LIN {X 0,Y 297.256,Z 379.745,A -85,B 0,C 180,E1 -16418.721,E2 -16418.721} C_VEL
LIN {X 0,Y 296.722,Z 381.976,A -85,B 0,C 180,E1 -16420.719,E2 -16420.719} C_VEL
LIN {X 0,Y 296.34,Z 383.559,A -85,B 0,C 180,E1 -16423.451,E2 -16423.451} C_VEL
LIN {X 0,Y 296.213,Z 383.714,A -85,B 0,C 180,E1 -16425.377,E2 -16425.377} C_VEL
LIN {X 0,Y 296.21,Z 383.053,A -85,B 0,C 180,E1 -16427.348,E2 -16427.348} C_VEL
LIN {X 0,Y 296.316,Z 381.493,A -85,B 0,C 180,E1 -16429.371,E2 -16429.371} C_VEL
LIN {X 0,Y 296.789,Z 378.032,A -85,B 0,C 180,E1 -16432,E2 -16432} C_VEL
LIN {X 0,Y 297.171,Z 374.788,A -85,B 0,C 180,E1 -16433.756,E2 -16433.756} C_VEL
LIN {X 0,Y 297.824,Z 369.2,A -85,B 0,C 180,E1 -16436.076,E2 -16436.076} C_VEL
LIN {X 0,Y 298.573,Z 363.535,A -85,B 0,C 180,E1 -16437.925,E2 -16437.925} C_VEL
LIN {X 0,Y 299.623,Z 356.033,A -85,B 0,C 180,E1 -16439.912,E2 -16439.912} C_VEL
LIN {X 0,Y 300.83,Z 347.311,A -85,B 0,C 180,E1 -16441.766,E2 -16441.766} C_VEL
LIN {X 0,Y 302.031,Z 337.923,A -85,B 0,C 180,E1 -16443.39,E2 -16443.39} C_VEL
LIN {X 0,Y 303.358,Z 327.596,A -85,B 0,C 180,E1 -16444.836,E2 -16444.836} C_VEL
LIN {X 0,Y 304.461,Z 317.398,A -85,B 0,C 180,E1 -16445.994,E2 -16445.994} C_VEL
LIN {X 0,Y 304.418,Z 313.925,A -85,B 0,C 180,E1 -16446.352,E2 -16446.352} C_VEL
LIN {X 0,Y 302.572,Z 302.571,A -85,B 0,C 180,E1 -16447.465,E2 -16447.465} C_VEL
LIN {X 0,Y 299.904,Z 289.87,A -85,B 0,C 180,E1 -16448.477,E2 -16448.477} C_VEL
LIN {X 0,Y 297.33,Z 278.987,A -85,B 0,C 180,E1 -16449.189,E2 -16449.189} C_VEL
LIN {X 0,Y 297.572,Z 275.868,A -85,B 0,C 180,E1 -16452.12,E2 -16452.12} C_VEL
LIN {X 0,Y 297.966,Z 271.492,A -85,B 0,C 180,E1 -16456.358,E2 -16456.358} C_VEL
LIN {X 0,Y 298.352,Z 267.326,A -85,B 0,C 180,E1 -16460.509,E2 -16460.509} C_VEL
LIN {X 0,Y 298.55,Z 266.296,A -85,B 0,C 180,E1 -16461.619,E2 -16461.619} C_VEL
LIN {X 0,Y 298.625,Z 266.288,A -85,B 0,C 180,E1 -16464.599,E2 -16464.599} C_VEL
LIN {X 0,Y 298.915,Z 266.253,A -85,B 0,C 180,E1 -16468.653,E2 -16468.653} C_VEL
LIN {X 0,Y 298.918,Z 266.248,A -85,B 0,C 180,E1 -16471.347,E2 -16471.347} C_VEL
LIN {X 0,Y 298.651,Z 266.281,A -85,B 0,C 180,E1 -16475.401,E2 -16475.401} C_VEL
LIN {X 0,Y 298.749,Z 266.273,A -85,B 0,C 180,E1 -16478.114,E2 -16478.114} C_VEL
LIN {X 0,Y 298.546,Z 266.299,A -85,B 0,C 180,E1 -16482.232,E2 -16482.232} C_VEL
LIN {X 0,Y 298.596,Z 266.288,A -85,B 0,C 180,E1 -16485.209,E2 -16485.209} C_VEL
LIN {X 0,Y 298.533,Z 266.295,A -85,B 0,C 180,E1 -16489.243,E2 -16489.243} C_VEL
LIN {X 0,Y 298.455,Z 266.308,A -85,B 0,C 180,E1 -16493.598,E2 -16493.598} C_VEL
LIN {X 0,Y 298.48,Z 266.301,A -85,B 0,C 180,E1 -16496.575,E2 -16496.575} C_VEL
LIN {X 0,Y 298.412,Z 266.312,A -85,B 0,C 180,E1 -16499.642,E2 -16499.642} C_VEL
LIN {X 0,Y 298.388,Z 266.314,A -85,B 0,C 180,E1 -16502.801,E2 -16502.801} C_VEL
LIN {X 0,Y 298.461,Z 266.305,A -85,B 0,C 180,E1 -16506.815,E2 -16506.815} C_VEL
LIN {X 0,Y 298.447,Z 266.307,A -85,B 0,C 180,E1 -16511.25,E2 -16511.25} C_VEL
LIN {X 0,Y 298.48,Z 266.303,A -85,B 0,C 180,E1 -16515.062,E2 -16515.062} C_VEL
LIN {X 0,Y 298.444,Z 266.309,A -85,B 0,C 180,E1 -16518.899,E2 -16518.899} C_VEL
LIN {X 0,Y 298.457,Z 266.309,A -85,B 0,C 180,E1 -16523.189,E2 -16523.189} C_VEL
LIN {X 0,Y 298.387,Z 266.314,A -85,B 0,C 180,E1 -16527.201,E2 -16527.201} C_VEL
LIN {X 0,Y 298.424,Z 266.307,A -85,B 0,C 180,E1 -16530.616,E2 -16530.616} C_VEL
LIN {X 0,Y 298.476,Z 266.302,A -85,B 0,C 180,E1 -16533.476,E2 -16533.476} C_VEL
LIN {X 0,Y 298.428,Z 266.312,A -85,B 0,C 180,E1 -16536.699,E2 -16536.699} C_VEL
LIN {X 0,Y 298.532,Z 266.3,A -85,B 0,C 180,E1 -16540.758,E2 -16540.758} C_VEL
LIN {X 0,Y 298.587,Z 266.288,A -85,B 0,C 180,E1 -16544.996,E2 -16544.996} C_VEL
LIN {X 0,Y 298.585,Z 266.286,A -85,B 0,C 180,E1 -16549.148,E2 -16549.148} C_VEL
LIN {X 0,Y 298.735,Z 266.27,A -85,B 0,C 180,E1 -16551.887,E2 -16551.887} C_VEL
LIN {X 0,Y 298.752,Z 266.266,A -85,B 0,C 180,E1 -16552.865,E2 -16552.865} C_VEL
LIN {X 0,Y 298.15,Z 266.346,A -85,B 0,C 180,E1 -16553.989,E2 -16553.989} C_VEL
LIN {X 0,Y 295.364,Z 266.697,A -85,B 0,C 180,E1 -16555.82,E2 -16555.82} C_VEL
LIN {X 0,Y 292.977,Z 266.993,A -85,B 0,C 180,E1 -16557.306,E2 -16557.306} C_VEL
LIN {X 0,Y 291.962,Z 267.117,A -85,B 0,C 180,E1 -16558.456,E2 -16558.456} C_VEL
LIN {X 0,Y 291.886,Z 267.124,A -85,B 0,C 180,E1 -16558.845,E2 -16558.845} C_VEL
LIN {X 0,Y 291.886,Z 267.122,A -85,B 0,C 180,E1 -16561.381,E2 -16561.381} C_VEL
LIN {X 0,Y 291.743,Z 267.139,A -85,B 0,C 180,E1 -16566.92,E2 -16566.92} C_VEL
LIN {X 0,Y 291.627,Z 267.158,A -85,B 0,C 180,E1 -16569.714,E2 -16569.714} C_VEL
LIN {X 0,Y 291.52,Z 267.173,A -85,B 0,C 180,E1 -16573.952,E2 -16573.952} C_VEL
LIN {X 0,Y 291.485,Z 267.172,A -85,B 0,C 180,E1 -16576.82,E2 -16576.82} C_VEL
LIN {X 0,Y 291.45,Z 267.181,A -85,B 0,C 180,E1 -16579.876,E2 -16579.876} C_VEL
LIN {X 0,Y 291.398,Z 267.185,A -85,B 0,C 180,E1 -16584.207,E2 -16584.207} C_VEL
LIN {X 0,Y 291.418,Z 267.184,A -85,B 0,C 180,E1 -16587.273,E2 -16587.273} C_VEL
LIN {X 0,Y 291.334,Z 267.193,A -85,B 0,C 180,E1 -16590.439,E2 -16590.439} C_VEL
LIN {X 0,Y 291.345,Z 267.194,A -85,B 0,C 180,E1 -16593.7,E2 -16593.7} C_VEL
LIN {X 0,Y 291.378,Z 267.192,A -85,B 0,C 180,E1 -16597.256,E2 -16597.256} C_VEL
LIN {X 0,Y 291.335,Z 267.194,A -85,B 0,C 180,E1 -16600.644,E2 -16600.644} C_VEL
LIN {X 0,Y 291.292,Z 267.199,A -85,B 0,C 180,E1 -16604.403,E2 -16604.403} C_VEL
LIN {X 0,Y 291.364,Z 267.287,A -85,B 0,C 180,E1 -16605.706,E2 -16605.706} C_VEL
LIN {X 0,Y 292.179,Z 271.679,A -85,B 0,C 180,E1 -16609.5,E2 -16609.5} C_VEL
LIN {X 0,Y 292.693,Z 275.227,A -85,B 0,C 180,E1 -16612.41,E2 -16612.41} C_VEL
LIN {X 0,Y 292.739,Z 278.292,A -85,B 0,C 180,E1 -16614.818,E2 -16614.818} C_VEL
LIN {X 0,Y 292.076,Z 282.608,A -85,B 0,C 180,E1 -16618.038,E2 -16618.038} C_VEL
LIN {X 0,Y 291.167,Z 289.009,A -85,B 0,C 180,E1 -16622.703,E2 -16622.703} C_VEL
LIN {X 0,Y 290.666,Z 294.198,A -85,B 0,C 180,E1 -16626.394,E2 -16626.394} C_VEL
LIN {X 0,Y 293.234,Z 308.199,A -85,B 0,C 180,E1 -16627.253,E2 -16627.253} C_VEL
LIN {X 0,Y 295.062,Z 320.852,A -85,B 0,C 180,E1 -16628.271,E2 -16628.271} C_VEL
LIN {X 0,Y 296.269,Z 331.555,A -85,B 0,C 180,E1 -16629.338,E2 -16629.338} C_VEL
LIN {X 0,Y 296.691,Z 338.172,A -85,B 0,C 180,E1 -16630.092,E2 -16630.092} C_VEL
LIN {X 0,Y 295.207,Z 348.791,A -85,B 0,C 180,E1 -16631.433,E2 -16631.433} C_VEL
LIN {X 0,Y 293.834,Z 359.224,A -85,B 0,C 180,E1 -16633.087,E2 -16633.087} C_VEL
LIN {X 0,Y 292.498,Z 369.063,A -85,B 0,C 180,E1 -16635.031,E2 -16635.031} C_VEL
LIN {X 0,Y 291.312,Z 377.393,A -85,B 0,C 180,E1 -16637.105,E2 -16637.105} C_VEL
LIN {X 0,Y 290.47,Z 384.109,A -85,B 0,C 180,E1 -16639.192,E2 -16639.192} C_VEL
LIN {X 0,Y 289.851,Z 390.238,A -85,B 0,C 180,E1 -16641.635,E2 -16641.635} C_VEL
LIN {X 0,Y 289.559,Z 394.197,A -85,B 0,C 180,E1 -16643.729,E2 -16643.729} C_VEL
LIN {X 0,Y 289.435,Z 397.097,A -85,B 0,C 180,E1 -16645.822,E2 -16645.822} C_VEL
LIN {X 0,Y 289.463,Z 398.458,A -85,B 0,C 180,E1 -16647.217,E2 -16647.217} C_VEL
LIN {X 0,Y 289.419,Z 399.41,A -85,B 0,C 180,E1 -16648.608,E2 -16648.608} C_VEL
LIN {X 0,Y 289.438,Z 399.968,A -85,B 0,C 180,E1 -16650,E2 -16650} C_VEL
LIN {X 0,Y 289.409,Z 400.104,A -85,B 0,C 180,E1 -16651.391,E2 -16651.391} C_VEL
LIN {X 0,Y 289.432,Z 399.814,A -85,B 0,C 180,E1 -16652.783,E2 -16652.783} C_VEL
LIN {X 0,Y 289.481,Z 398.063,A -85,B 0,C 180,E1 -16655.573,E2 -16655.573} C_VEL
LIN {X 0,Y 289.638,Z 396.572,A -85,B 0,C 180,E1 -16656.968,E2 -16656.968} C_VEL
LIN {X 0,Y 290.082,Z 393.523,A -85,B 0,C 180,E1 -16659.06,E2 -16659.06} C_VEL
LIN {X 0,Y 290.789,Z 389.449,A -85,B 0,C 180,E1 -16661.148,E2 -16661.148} C_VEL
LIN {X 0,Y 292.006,Z 383.239,A -85,B 0,C 180,E1 -16663.571,E2 -16663.571} C_VEL
LIN {X 0,Y 293.614,Z 376.515,A -85,B 0,C 180,E1 -16665.621,E2 -16665.621} C_VEL
LIN {X 0,Y 295.014,Z 369.133,A -85,B 0,C 180,E1 -16667.467,E2 -16667.467} C_VEL
LIN {X 0,Y 296.963,Z 359.815,A -85,B 0,C 180,E1 -16669.349,E2 -16669.349} C_VEL
LIN {X 0,Y 299.12,Z 349.497,A -85,B 0,C 180,E1 -16670.996,E2 -16670.996} C_VEL
LIN {X 0,Y 300.497,Z 342.181,A -85,B 0,C 180,E1 -16671.975,E2 -16671.975} C_VEL
LIN {X 0,Y 300.225,Z 332.312,A -85,B 0,C 180,E1 -16673.273,E2 -16673.273} C_VEL
LIN {X 0,Y 299.063,Z 321.612,A -85,B 0,C 180,E1 -16674.529,E2 -16674.529} C_VEL
LIN {X 0,Y 297.128,Z 311.576,A -85,B 0,C 180,E1 -16675.605,E2 -16675.605} C_VEL
LIN {X 0,Y 293.476,Z 298.869,A -85,B 0,C 180,E1 -16676.88,E2 -16676.88} C_VEL
LIN {X 0,Y 291.642,Z 293.187,A -85,B 0,C 180,E1 -16677.401,E2 -16677.401} C_VEL
LIN {X 0,Y 291.589,Z 292.614,A -85,B 0,C 180,E1 -16677.494,E2 -16677.494} C_VEL
LIN {X 0,Y 292.14,Z 288.963,A -85,B 0,C 180,E1 -16680.343,E2 -16680.343} C_VEL
LIN {X 0,Y 292.807,Z 285.096,A -85,B 0,C 180,E1 -16683.507,E2 -16683.507} C_VEL
LIN {X 0,Y 293.161,Z 282.887,A -85,B 0,C 180,E1 -16685.402,E2 -16685.402} C_VEL
LIN {X 0,Y 293.236,Z 279.487,A -85,B 0,C 180,E1 -16688.545,E2 -16688.545} C_VEL
LIN {X 0,Y 292.811,Z 275.93,A -85,B 0,C 180,E1 -16692.224,E2 -16692.224} C_VEL
LIN {X 0,Y 292.299,Z 272.574,A -85,B 0,C 180,E1 -16696.162,E2 -16696.162} C_VEL
LIN {X 0,Y 291.787,Z 269.447,A -85,B 0,C 180,E1 -16700.42,E2 -16700.42} C_VEL
LIN {X 0,Y 291.524,Z 267.869,A -85,B 0,C 180,E1 -16702.935,E2 -16702.935} C_VEL
LIN {X 0,Y 291.389,Z 267.189,A -85,B 0,C 180,E1 -16705.087,E2 -16705.087} C_VEL
LIN {X 0,Y 291.371,Z 267.192,A -85,B 0,C 180,E1 -16707.949,E2 -16707.949} C_VEL
LIN {X 0,Y 291.38,Z 267.189,A -85,B 0,C 180,E1 -16711.157,E2 -16711.157} C_VEL
LIN {X 0,Y 291.415,Z 267.187,A -85,B 0,C 180,E1 -16714.27,E2 -16714.27} C_VEL
LIN {X 0,Y 291.378,Z 267.19,A -85,B 0,C 180,E1 -16717.298,E2 -16717.298} C_VEL
LIN {X 0,Y 291.455,Z 267.181,A -85,B 0,C 180,E1 -16720.268,E2 -16720.268} C_VEL
LIN {X 0,Y 291.537,Z 267.172,A -85,B 0,C 180,E1 -16724.633,E2 -16724.633} C_VEL
LIN {X 0,Y 291.532,Z 267.171,A -85,B 0,C 180,E1 -16728.879,E2 -16728.879} C_VEL
LIN {X 0,Y 291.704,Z 267.151,A -85,B 0,C 180,E1 -16731.687,E2 -16731.687} C_VEL
LIN {X 0,Y 291.625,Z 267.158,A -85,B 0,C 180,E1 -16734.467,E2 -16734.467} C_VEL
LIN {X 0,Y 291.884,Z 267.126,A -85,B 0,C 180,E1 -16738.619,E2 -16738.619} C_VEL
LIN {X 0,Y 292.013,Z 267.48,A -85,B 0,C 180,E1 -16739.998,E2 -16739.998} C_VEL
LIN {X 0,Y 292.074,Z 269.02,A -85,B 0,C 180,E1 -16742.757,E2 -16742.757} C_VEL
LIN {X 0,Y 292.277,Z 271.603,A -85,B 0,C 180,E1 -16746.904,E2 -16746.904} C_VEL
LIN {X 0,Y 292.339,Z 273.56,A -85,B 0,C 180,E1 -16749.722,E2 -16749.722} C_VEL
LIN {X 0,Y 291.837,Z 276.856,A -85,B 0,C 180,E1 -16753.933,E2 -16753.933} C_VEL
LIN {X 0,Y 291.452,Z 279.266,A -85,B 0,C 180,E1 -16756.818,E2 -16756.818} C_VEL
LIN {X 0,Y 291.228,Z 280.798,A -85,B 0,C 180,E1 -16758.6,E2 -16758.6} C_VEL
LIN {X 0,Y 292.241,Z 283.889,A -85,B 0,C 180,E1 -16758.897,E2 -16758.897} C_VEL
LIN {X 0,Y 296.303,Z 294.553,A -85,B 0,C 180,E1 -16760.086,E2 -16760.086} C_VEL
LIN {X 0,Y 299.322,Z 304.767,A -85,B 0,C 180,E1 -16761.272,E2 -16761.272} C_VEL
LIN {X 0,Y 301.593,Z 316.345,A -85,B 0,C 180,E1 -16762.716,E2 -16762.716} C_VEL
LIN {X 0,Y 302.352,Z 322.44,A -85,B 0,C 180,E1 -16763.539,E2 -16763.539} C_VEL
LIN {X 0,Y 300.502,Z 333.167,A -85,B 0,C 180,E1 -16764.894,E2 -16764.894} C_VEL
LIN {X 0,Y 298.4,Z 343.82,A -85,B 0,C 180,E1 -16766.581,E2 -16766.581} C_VEL
LIN {X 0,Y 296.514,Z 352.555,A -85,B 0,C 180,E1 -16768.295,E2 -16768.295} C_VEL
LIN {X 0,Y 294.957,Z 359.715,A -85,B 0,C 180,E1 -16770.022,E2 -16770.022} C_VEL
LIN {X 0,Y 293.128,Z 367.333,A -85,B 0,C 180,E1 -16772.313,E2 -16772.313} C_VEL
LIN {X 0,Y 291.934,Z 372.454,A -85,B 0,C 180,E1 -16774.268,E2 -16774.268} C_VEL
LIN {X 0,Y 291.015,Z 376.512,A -85,B 0,C 180,E1 -16776.223,E2 -16776.223} C_VEL
LIN {X 0,Y 290.349,Z 379.544,A -85,B 0,C 180,E1 -16778.112,E2 -16778.112} C_VEL
LIN {X 0,Y 290.043,Z 380.865,A -85,B 0,C 180,E1 -16779.161,E2 -16779.161} C_VEL
LIN {X 0,Y 289.559,Z 382.745,A -85,B 0,C 180,E1 -16781.202,E2 -16781.202} C_VEL
LIN {X 0,Y 289.272,Z 383.745,A -85,B 0,C 180,E1 -16783.21,E2 -16783.21} C_VEL
LIN {X 0,Y 289.136,Z 383.93,A -85,B 0,C 180,E1 -16785.18,E2 -16785.18} C_VEL
LIN {X 0,Y 289.1,Z 383.357,A -85,B 0,C 180,E1 -16787.105,E2 -16787.105} C_VEL
LIN {X 0,Y 289.291,Z 381.069,A -85,B 0,C 180,E1 -16789.926,E2 -16789.926} C_VEL
LIN {X 0,Y 289.666,Z 378.543,A -85,B 0,C 180,E1 -16791.836,E2 -16791.836} C_VEL
LIN {X 0,Y 290.236,Z 373.662,A -85,B 0,C 180,E1 -16794.469,E2 -16794.469} C_VEL
LIN {X 0,Y 290.917,Z 368.352,A -85,B 0,C 180,E1 -16796.596,E2 -16796.596} C_VEL
LIN {X 0,Y 291.897,Z 361.234,A -85,B 0,C 180,E1 -16798.826,E2 -16798.826} C_VEL
LIN {X 0,Y 293.127,Z 352.689,A -85,B 0,C 180,E1 -16800.955,E2 -16800.955} C_VEL
LIN {X 0,Y 294.342,Z 343.846,A -85,B 0,C 180,E1 -16802.724,E2 -16802.724} C_VEL
LIN {X 0,Y 295.724,Z 333.278,A -85,B 0,C 180,E1 -16804.427,E2 -16804.427} C_VEL
LIN {X 0,Y 297.002,Z 323.285,A -85,B 0,C 180,E1 -16805.724,E2 -16805.724} C_VEL
LIN {X 0,Y 297.663,Z 316.026,A -85,B 0,C 180,E1 -16806.521,E2 -16806.521} C_VEL
LIN {X 0,Y 295.95,Z 304.983,A -85,B 0,C 180,E1 -16807.67,E2 -16807.67} C_VEL
LIN {X 0,Y 293.272,Z 291.758,A -85,B 0,C 180,E1 -16808.796,E2 -16808.796} C_VEL
LIN {X 0,Y 290.272,Z 279.187,A -85,B 0,C 180,E1 -16809.633,E2 -16809.633} C_VEL
LIN {X 0,Y 290.557,Z 275.578,A -85,B 0,C 180,E1 -16813.127,E2 -16813.127} C_VEL
LIN {X 0,Y 290.879,Z 272.648,A -85,B 0,C 180,E1 -16816.019,E2 -16816.019} C_VEL
LIN {X 0,Y 291.278,Z 268.444,A -85,B 0,C 180,E1 -16820.277,E2 -16820.277} C_VEL
LIN {X 0,Y 291.504,Z 267.174,A -85,B 0,C 180,E1 -16821.683,E2 -16821.683} C_VEL
LIN {X 0,Y 291.59,Z 267.163,A -85,B 0,C 180,E1 -16824.468,E2 -16824.468} C_VEL
LIN {X 0,Y 291.881,Z 267.129,A -85,B 0,C 180,E1 -16828.621,E2 -16828.621} C_VEL
LIN {X 0,Y 291.884,Z 267.124,A -85,B 0,C 180,E1 -16831.38,E2 -16831.38} C_VEL
LIN {X 0,Y 291.736,Z 267.144,A -85,B 0,C 180,E1 -16836.918,E2 -16836.918} C_VEL
LIN {X 0,Y 291.62,Z 267.158,A -85,B 0,C 180,E1 -16839.712,E2 -16839.712} C_VEL
LIN {X 0,Y 291.513,Z 267.173,A -85,B 0,C 180,E1 -16843.951,E2 -16843.951} C_VEL
LIN {X 0,Y 291.477,Z 267.174,A -85,B 0,C 180,E1 -16846.818,E2 -16846.818} C_VEL
LIN {X 0,Y 291.442,Z 267.182,A -85,B 0,C 180,E1 -16849.876,E2 -16849.876} C_VEL
LIN {X 0,Y 291.413,Z 267.185,A -85,B 0,C 180,E1 -16854.204,E2 -16854.204} C_VEL
LIN {X 0,Y 291.413,Z 267.181,A -85,B 0,C 180,E1 -16857.272,E2 -16857.272} C_VEL
LIN {X 0,Y 291.329,Z 267.193,A -85,B 0,C 180,E1 -16860.437,E2 -16860.437} C_VEL
LIN {X 0,Y 291.336,Z 267.197,A -85,B 0,C 180,E1 -16863.699,E2 -16863.699} C_VEL
LIN {X 0,Y 291.396,Z 267.187,A -85,B 0,C 180,E1 -16867.262,E2 -16867.262} C_VEL
LIN {X 0,Y 291.397,Z 267.181,A -85,B 0,C 180,E1 -16870.631,E2 -16870.631} C_VEL
LIN {X 0,Y 291.397,Z 267.182,A -85,B 0,C 180,E1 -16874.38,E2 -16874.38} C_VEL
LIN {X 0,Y 291.38,Z 267.187,A -85,B 0,C 180,E1 -16878.392,E2 -16878.392} C_VEL
LIN {X 0,Y 291.371,Z 267.192,A -85,B 0,C 180,E1 -16881.164,E2 -16881.164} C_VEL
LIN {X 0,Y 291.377,Z 267.187,A -85,B 0,C 180,E1 -16884.631,E2 -16884.631} C_VEL
LIN {X 0,Y 291.363,Z 267.184,A -85,B 0,C 180,E1 -16887.952,E2 -16887.952} C_VEL
LIN {X 0,Y 291.375,Z 267.188,A -85,B 0,C 180,E1 -16891.16,E2 -16891.16} C_VEL
LIN {X 0,Y 291.409,Z 267.182,A -85,B 0,C 180,E1 -16894.273,E2 -16894.273} C_VEL
LIN {X 0,Y 291.374,Z 267.189,A -85,B 0,C 180,E1 -16897.301,E2 -16897.301} C_VEL
LIN {X 0,Y 291.451,Z 267.179,A -85,B 0,C 180,E1 -16900.272,E2 -16900.272} C_VEL
LIN {X 0,Y 291.534,Z 267.169,A -85,B 0,C 180,E1 -16904.636,E2 -16904.636} C_VEL
LIN {X 0,Y 291.529,Z 267.166,A -85,B 0,C 180,E1 -16908.882,E2 -16908.882} C_VEL
LIN {X 0,Y 291.682,Z 267.147,A -85,B 0,C 180,E1 -16911.689,E2 -16911.689} C_VEL
LIN {X 0,Y 291.622,Z 267.161,A -85,B 0,C 180,E1 -16914.47,E2 -16914.47} C_VEL
LIN {X 0,Y 291.886,Z 267.124,A -85,B 0,C 180,E1 -16918.845,E2 -16918.845} C_VEL
LIN {X 0,Y 291.563,Z 267.164,A -85,B 0,C 180,E1 -16919.616,E2 -16919.616} C_VEL
LIN {X 0,Y 289.526,Z 267.419,A -85,B 0,C 180,E1 -16921.126,E2 -16921.126} C_VEL
LIN {X 0,Y 285.64,Z 267.9,A -85,B 0,C 180,E1 -16923.39,E2 -16923.39} C_VEL
LIN {X 0,Y 284.593,Z 268.028,A -85,B 0,C 180,E1 -16924.573,E2 -16924.573} C_VEL
LIN {X 0,Y 284.53,Z 268.034,A -85,B 0,C 180,E1 -16924.973,E2 -16924.973} C_VEL
LIN {X 0,Y 284.695,Z 268.016,A -85,B 0,C 180,E1 -16927.092,E2 -16927.092} C_VEL
LIN {X 0,Y 284.565,Z 268.039,A -85,B 0,C 180,E1 -16929.957,E2 -16929.957} C_VEL
LIN {X 0,Y 284.477,Z 268.048,A -85,B 0,C 180,E1 -16934.305,E2 -16934.305} C_VEL
LIN {X 0,Y 284.423,Z 268.052,A -85,B 0,C 180,E1 -16937.25,E2 -16937.25} C_VEL
LIN {X 0,Y 284.378,Z 268.059,A -85,B 0,C 180,E1 -16940.244,E2 -16940.244} C_VEL
LIN {X 0,Y 284.368,Z 268.063,A -85,B 0,C 180,E1 -16943.876,E2 -16943.876} C_VEL
LIN {X 0,Y 284.394,Z 268.058,A -85,B 0,C 180,E1 -16947.174,E2 -16947.174} C_VEL
LIN {X 0,Y 284.294,Z 268.073,A -85,B 0,C 180,E1 -16951.276,E2 -16951.276} C_VEL
LIN {X 0,Y 284.342,Z 268.067,A -85,B 0,C 180,E1 -16955.349,E2 -16955.349} C_VEL
LIN {X 0,Y 284.314,Z 268.068,A -85,B 0,C 180,E1 -16958.17,E2 -16958.17} C_VEL
LIN {X 0,Y 284.271,Z 268.073,A -85,B 0,C 180,E1 -16962.126,E2 -16962.126} C_VEL
LIN {X 0,Y 284.318,Z 268.271,A -85,B 0,C 180,E1 -16965.577,E2 -16965.577} C_VEL
LIN {X 0,Y 284.93,Z 271.255,A -85,B 0,C 180,E1 -16968.244,E2 -16968.244} C_VEL
LIN {X 0,Y 285.603,Z 275.711,A -85,B 0,C 180,E1 -16972.035,E2 -16972.035} C_VEL
LIN {X 0,Y 285.72,Z 278.465,A -85,B 0,C 180,E1 -16974.266,E2 -16974.266} C_VEL
LIN {X 0,Y 285.222,Z 282.234,A -85,B 0,C 180,E1 -16977.174,E2 -16977.174} C_VEL
LIN {X 0,Y 284.22,Z 288.642,A -85,B 0,C 180,E1 -16981.978,E2 -16981.978} C_VEL
LIN {X 0,Y 283.649,Z 294.031,A -85,B 0,C 180,E1 -16985.918,E2 -16985.918} C_VEL
LIN {X 0,Y 286.123,Z 307.348,A -85,B 0,C 180,E1 -16986.745,E2 -16986.745} C_VEL
LIN {X 0,Y 288.089,Z 320.565,A -85,B 0,C 180,E1 -16987.838,E2 -16987.838} C_VEL
LIN {X 0,Y 289.345,Z 331.936,A -85,B 0,C 180,E1 -16989.006,E2 -16989.006} C_VEL
LIN {X 0,Y 289.749,Z 338.469,A -85,B 0,C 180,E1 -16989.779,E2 -16989.779} C_VEL
LIN {X 0,Y 288.104,Z 350.156,A -85,B 0,C 180,E1 -16991.327,E2 -16991.327} C_VEL
LIN {X 0,Y 286.817,Z 359.652,A -85,B 0,C 180,E1 -16992.9,E2 -16992.9} C_VEL
LIN {X 0,Y 285.606,Z 368.348,A -85,B 0,C 180,E1 -16994.661,E2 -16994.661} C_VEL
LIN {X 0,Y 284.371,Z 376.786,A -85,B 0,C 180,E1 -16996.785,E2 -16996.785} C_VEL
LIN {X 0,Y 283.462,Z 383.575,A -85,B 0,C 180,E1 -16998.922,E2 -16998.922} C_VEL
LIN {X 0,Y 282.799,Z 389.798,A -85,B 0,C 180,E1 -17001.425,E2 -17001.425} C_VEL
LIN {X 0,Y 282.492,Z 393.817,A -85,B 0,C 180,E1 -17003.572,E2 -17003.572} C_VEL
LIN {X 0,Y 282.342,Z 396.767,A -85,B 0,C 180,E1 -17005.717,E2 -17005.717} C_VEL
LIN {X 0,Y 282.369,Z 398.165,A -85,B 0,C 180,E1 -17007.147,E2 -17007.147} C_VEL
LIN {X 0,Y 282.342,Z 399.144,A -85,B 0,C 180,E1 -17008.573,E2 -17008.573} C_VEL
LIN {X 0,Y 282.358,Z 399.727,A -85,B 0,C 180,E1 -17010,E2 -17010} C_VEL
LIN {X 0,Y 282.333,Z 399.908,A -85,B 0,C 180,E1 -17011.426,E2 -17011.426} C_VEL
LIN {X 0,Y 282.338,Z 399.648,A -85,B 0,C 180,E1 -17012.853,E2 -17012.853} C_VEL
LIN {X 0,Y 282.391,Z 397.95,A -85,B 0,C 180,E1 -17015.713,E2 -17015.713} C_VEL
LIN {X 0,Y 282.579,Z 396.51,A -85,B 0,C 180,E1 -17017.143,E2 -17017.143} C_VEL
LIN {X 0,Y 283.057,Z 393.517,A -85,B 0,C 180,E1 -17019.287,E2 -17019.287} C_VEL
LIN {X 0,Y 283.816,Z 389.503,A -85,B 0,C 180,E1 -17021.425,E2 -17021.425} C_VEL
LIN {X 0,Y 285.108,Z 383.389,A -85,B 0,C 180,E1 -17023.906,E2 -17023.906} C_VEL
LIN {X 0,Y 286.796,Z 376.739,A -85,B 0,C 180,E1 -17026.002,E2 -17026.002} C_VEL
LIN {X 0,Y 288.634,Z 367.851,A -85,B 0,C 180,E1 -17028.261,E2 -17028.261} C_VEL
LIN {X 0,Y 290.753,Z 358.408,A -85,B 0,C 180,E1 -17030.147,E2 -17030.147} C_VEL
LIN {X 0,Y 293.043,Z 347.904,A -85,B 0,C 180,E1 -17031.822,E2 -17031.822} C_VEL
LIN {X 0,Y 294.002,Z 341.921,A -85,B 0,C 180,E1 -17032.649,E2 -17032.649} C_VEL
LIN {X 0,Y 293.528,Z 330.262,A -85,B 0,C 180,E1 -17034.213,E2 -17034.213} C_VEL
LIN {X 0,Y 291.859,Z 317.94,A -85,B 0,C 180,E1 -17035.685,E2 -17035.685} C_VEL
LIN {X 0,Y 288.827,Z 305.475,A -85,B 0,C 180,E1 -17037.078,E2 -17037.078} C_VEL
LIN {X 0,Y 285.489,Z 295.291,A -85,B 0,C 180,E1 -17038.136,E2 -17038.136} C_VEL
LIN {X 0,Y 284.738,Z 292.405,A -85,B 0,C 180,E1 -17038.407,E2 -17038.407} C_VEL
LIN {X 0,Y 285.639,Z 287.112,A -85,B 0,C 180,E1 -17042.771,E2 -17042.771} C_VEL
LIN {X 0,Y 286.199,Z 283.326,A -85,B 0,C 180,E1 -17046.11,E2 -17046.11} C_VEL
LIN {X 0,Y 286.277,Z 281.113,A -85,B 0,C 180,E1 -17048.223,E2 -17048.223} C_VEL
LIN {X 0,Y 285.913,Z 277.91,A -85,B 0,C 180,E1 -17051.58,E2 -17051.58} C_VEL
LIN {X 0,Y 285.426,Z 274.532,A -85,B 0,C 180,E1 -17055.565,E2 -17055.565} C_VEL
LIN {X 0,Y 284.915,Z 271.383,A -85,B 0,C 180,E1 -17059.877,E2 -17059.877} C_VEL
LIN {X 0,Y 284.52,Z 269.091,A -85,B 0,C 180,E1 -17063.64,E2 -17063.64} C_VEL
LIN {X 0,Y 284.34,Z 268.198,A -85,B 0,C 180,E1 -17065.353,E2 -17065.353} C_VEL
LIN {X 0,Y 284.294,Z 268.072,A -85,B 0,C 180,E1 -17068.724,E2 -17068.724} C_VEL
LIN {X 0,Y 284.396,Z 268.06,A -85,B 0,C 180,E1 -17072.825,E2 -17072.825} C_VEL
LIN {X 0,Y 284.364,Z 268.065,A -85,B 0,C 180,E1 -17076.705,E2 -17076.705} C_VEL
LIN {X 0,Y 284.4,Z 268.059,A -85,B 0,C 180,E1 -17081.26,E2 -17081.26} C_VEL
LIN {X 0,Y 284.474,Z 268.052,A -85,B 0,C 180,E1 -17084.468,E2 -17084.468} C_VEL
LIN {X 0,Y 284.484,Z 268.05,A -85,B 0,C 180,E1 -17088.6,E2 -17088.6} C_VEL
LIN {X 0,Y 284.654,Z 268.029,A -85,B 0,C 180,E1 -17091.479,E2 -17091.479} C_VEL
LIN {X 0,Y 284.596,Z 268.034,A -85,B 0,C 180,E1 -17094.33,E2 -17094.33} C_VEL
LIN {X 0,Y 284.739,Z 268.017,A -85,B 0,C 180,E1 -17097.169,E2 -17097.169} C_VEL
LIN {X 0,Y 284.883,Z 268.286,A -85,B 0,C 180,E1 -17098.585,E2 -17098.585} C_VEL
LIN {X 0,Y 285.12,Z 269.678,A -85,B 0,C 180,E1 -17101.411,E2 -17101.411} C_VEL
LIN {X 0,Y 285.278,Z 272.935,A -85,B 0,C 180,E1 -17106.908,E2 -17106.908} C_VEL
LIN {X 0,Y 285.327,Z 274.985,A -85,B 0,C 180,E1 -17109.927,E2 -17109.927} C_VEL
LIN {X 0,Y 284.973,Z 277.165,A -85,B 0,C 180,E1 -17112.822,E2 -17112.822} C_VEL
LIN {X 0,Y 284.599,Z 279.509,A -85,B 0,C 180,E1 -17115.76,E2 -17115.76} C_VEL
LIN {X 0,Y 284.327,Z 281.063,A -85,B 0,C 180,E1 -17117.624,E2 -17117.624} C_VEL
LIN {X 0,Y 285.381,Z 284.267,A -85,B 0,C 180,E1 -17117.973,E2 -17117.973} C_VEL
LIN {X 0,Y 289.433,Z 294.425,A -85,B 0,C 180,E1 -17119.18,E2 -17119.18} C_VEL
LIN {X 0,Y 292.846,Z 305.93,A -85,B 0,C 180,E1 -17120.602,E2 -17120.602} C_VEL
LIN {X 0,Y 295.002,Z 316.877,A -85,B 0,C 180,E1 -17122.036,E2 -17122.036} C_VEL
LIN {X 0,Y 295.819,Z 324.286,A -85,B 0,C 180,E1 -17123.077,E2 -17123.077} C_VEL
LIN {X 0,Y 293.719,Z 335.646,A -85,B 0,C 180,E1 -17124.601,E2 -17124.601} C_VEL
LIN {X 0,Y 291.696,Z 345.269,A -85,B 0,C 180,E1 -17126.211,E2 -17126.211} C_VEL
LIN {X 0,Y 289.567,Z 354.379,A -85,B 0,C 180,E1 -17128.114,E2 -17128.114} C_VEL
LIN {X 0,Y 287.808,Z 361.793,A -85,B 0,C 180,E1 -17130.037,E2 -17130.037} C_VEL
LIN {X 0,Y 286.035,Z 368.807,A -85,B 0,C 180,E1 -17132.301,E2 -17132.301} C_VEL
LIN {X 0,Y 284.694,Z 374.307,A -85,B 0,C 180,E1 -17134.593,E2 -17134.593} C_VEL
LIN {X 0,Y 283.85,Z 377.755,A -85,B 0,C 180,E1 -17136.455,E2 -17136.455} C_VEL
LIN {X 0,Y 283.187,Z 380.448,A -85,B 0,C 180,E1 -17138.345,E2 -17138.345} C_VEL
LIN {X 0,Y 282.634,Z 382.441,A -85,B 0,C 180,E1 -17140.277,E2 -17140.277} C_VEL
LIN {X 0,Y 282.306,Z 383.686,A -85,B 0,C 180,E1 -17142.231,E2 -17142.231} C_VEL
LIN {X 0,Y 282.075,Z 384.16,A -85,B 0,C 180,E1 -17144.234,E2 -17144.234} C_VEL
LIN {X 0,Y 282.012,Z 383.853,A -85,B 0,C 180,E1 -17146.275,E2 -17146.275} C_VEL
LIN {X 0,Y 282.029,Z 382.69,A -85,B 0,C 180,E1 -17148.378,E2 -17148.378} C_VEL
LIN {X 0,Y 282.291,Z 380.595,A -85,B 0,C 180,E1 -17150.511,E2 -17150.511} C_VEL
LIN {X 0,Y 282.729,Z 377.437,A -85,B 0,C 180,E1 -17152.694,E2 -17152.694} C_VEL
LIN {X 0,Y 283.382,Z 372.369,A -85,B 0,C 180,E1 -17155.222,E2 -17155.222} C_VEL
LIN {X 0,Y 284.226,Z 365.982,A -85,B 0,C 180,E1 -17157.637,E2 -17157.637} C_VEL
LIN {X 0,Y 285.184,Z 359.408,A -85,B 0,C 180,E1 -17159.598,E2 -17159.598} C_VEL
LIN {X 0,Y 286.473,Z 350.732,A -85,B 0,C 180,E1 -17161.678,E2 -17161.678} C_VEL
LIN {X 0,Y 287.798,Z 341.157,A -85,B 0,C 180,E1 -17163.535,E2 -17163.535} C_VEL
LIN {X 0,Y 289.112,Z 331.728,A -85,B 0,C 180,E1 -17165.017,E2 -17165.017} C_VEL
LIN {X 0,Y 290.539,Z 320.094,A -85,B 0,C 180,E1 -17166.478,E2 -17166.478} C_VEL
LIN {X 0,Y 290.778,Z 316.872,A -85,B 0,C 180,E1 -17166.837,E2 -17166.837} C_VEL
LIN {X 0,Y 289.04,Z 305.673,A -85,B 0,C 180,E1 -17168.048,E2 -17168.048} C_VEL
LIN {X 0,Y 286.385,Z 292.575,A -85,B 0,C 180,E1 -17169.208,E2 -17169.208} C_VEL
LIN {X 0,Y 283.246,Z 279.387,A -85,B 0,C 180,E1 -17170.108,E2 -17170.108} C_VEL
LIN {X 0,Y 283.591,Z 275.274,A -85,B 0,C 180,E1 -17174.181,E2 -17174.181} C_VEL
LIN {X 0,Y 283.887,Z 272.39,A -85,B 0,C 180,E1 -17177.127,E2 -17177.127} C_VEL
LIN {X 0,Y 284.46,Z 268.052,A -85,B 0,C 180,E1 -17181.717,E2 -17181.717} C_VEL
LIN {X 0,Y 284.554,Z 268.038,A -85,B 0,C 180,E1 -17184.331,E2 -17184.331} C_VEL
LIN {X 0,Y 284.847,Z 268.006,A -85,B 0,C 180,E1 -17188.586,E2 -17188.586} C_VEL
LIN {X 0,Y 284.85,Z 268.001,A -85,B 0,C 180,E1 -17191.414,E2 -17191.414} C_VEL
LIN {X 0,Y 284.688,Z 268.022,A -85,B 0,C 180,E1 -17197.09,E2 -17197.09} C_VEL
LIN {X 0,Y 284.557,Z 268.039,A -85,B 0,C 180,E1 -17199.956,E2 -17199.956} C_VEL
LIN {X 0,Y 284.472,Z 268.051,A -85,B 0,C 180,E1 -17204.303,E2 -17204.303} C_VEL
LIN {X 0,Y 284.416,Z 268.053,A -85,B 0,C 180,E1 -17207.249,E2 -17207.249} C_VEL
LIN {X 0,Y 284.372,Z 268.063,A -85,B 0,C 180,E1 -17210.243,E2 -17210.243} C_VEL
LIN {X 0,Y 284.375,Z 268.064,A -85,B 0,C 180,E1 -17213.883,E2 -17213.883} C_VEL
LIN {X 0,Y 284.388,Z 268.056,A -85,B 0,C 180,E1 -17217.174,E2 -17217.174} C_VEL
LIN {X 0,Y 284.288,Z 268.07,A -85,B 0,C 180,E1 -17221.275,E2 -17221.275} C_VEL
LIN {X 0,Y 284.353,Z 268.065,A -85,B 0,C 180,E1 -17225.355,E2 -17225.355} C_VEL
LIN {X 0,Y 284.328,Z 268.064,A -85,B 0,C 180,E1 -17228.166,E2 -17228.166} C_VEL
LIN {X 0,Y 284.335,Z 268.059,A -85,B 0,C 180,E1 -17232.142,E2 -17232.142} C_VEL
LIN {X 0,Y 284.344,Z 268.062,A -85,B 0,C 180,E1 -17236.209,E2 -17236.209} C_VEL
LIN {X 0,Y 284.343,Z 268.064,A -85,B 0,C 180,E1 -17240.014,E2 -17240.014} C_VEL
LIN {X 0,Y 284.344,Z 268.063,A -85,B 0,C 180,E1 -17243.618,E2 -17243.618} C_VEL
LIN {X 0,Y 284.299,Z 268.067,A -85,B 0,C 180,E1 -17247.191,E2 -17247.191} C_VEL
LIN {X 0,Y 284.351,Z 268.056,A -85,B 0,C 180,E1 -17250.377,E2 -17250.377} C_VEL
LIN {X 0,Y 284.37,Z 268.059,A -85,B 0,C 180,E1 -17253.588,E2 -17253.588} C_VEL
LIN {X 0,Y 284.359,Z 268.065,A -85,B 0,C 180,E1 -17256.708,E2 -17256.708} C_VEL
LIN {X 0,Y 284.397,Z 268.057,A -85,B 0,C 180,E1 -17261.263,E2 -17261.263} C_VEL
LIN {X 0,Y 284.472,Z 268.048,A -85,B 0,C 180,E1 -17264.471,E2 -17264.471} C_VEL
LIN {X 0,Y 284.481,Z 268.044,A -85,B 0,C 180,E1 -17268.603,E2 -17268.603} C_VEL
LIN {X 0,Y 284.633,Z 268.024,A -85,B 0,C 180,E1 -17271.482,E2 -17271.482} C_VEL
LIN {X 0,Y 284.592,Z 268.036,A -85,B 0,C 180,E1 -17274.333,E2 -17274.333} C_VEL
LIN {X 0,Y 284.85,Z 268.001,A -85,B 0,C 180,E1 -17278.848,E2 -17278.848} C_VEL
LIN {X 0,Y 284.852,Z 267.998,A -85,B 0,C 180,E1 -17281.415,E2 -17281.415} C_VEL
LIN {X 0,Y 284.53,Z 268.034,A -85,B 0,C 180,E1 -17284.973,E2 -17284.973} C_VEL
LIN {X 0,Y 283.919,Z 268.116,A -85,B 0,C 180,E1 -17286.157,E2 -17286.157} C_VEL
LIN {X 0,Y 281.064,Z 268.474,A -85,B 0,C 180,E1 -17288.085,E2 -17288.085} C_VEL
LIN {X 0,Y 278.597,Z 268.78,A -85,B 0,C 180,E1 -17289.65,E2 -17289.65} C_VEL
LIN {X 0,Y 277.526,Z 268.913,A -85,B 0,C 180,E1 -17290.864,E2 -17290.864} C_VEL
LIN {X 0,Y 277.435,Z 268.924,A -85,B 0,C 180,E1 -17291.276,E2 -17291.276} C_VEL
LIN {X 0,Y 277.434,Z 268.927,A -85,B 0,C 180,E1 -17295.718,E2 -17295.718} C_VEL
LIN {X 0,Y 277.344,Z 268.934,A -85,B 0,C 180,E1 -17300.351,E2 -17300.351} C_VEL
LIN {X 0,Y 277.318,Z 268.94,A -85,B 0,C 180,E1 -17304.171,E2 -17304.171} C_VEL
LIN {X 0,Y 277.323,Z 268.94,A -85,B 0,C 180,E1 -17307.505,E2 -17307.505} C_VEL
LIN {X 0,Y 277.273,Z 268.945,A -85,B 0,C 180,E1 -17310.483,E2 -17310.483} C_VEL
LIN {X 0,Y 277.248,Z 268.948,A -85,B 0,C 180,E1 -17313.897,E2 -17313.897} C_VEL
LIN {X 0,Y 277.27,Z 268.949,A -85,B 0,C 180,E1 -17317.471,E2 -17317.471} C_VEL
LIN {X 0,Y 277.212,Z 268.956,A -85,B 0,C 180,E1 -17321.238,E2 -17321.238} C_VEL
LIN {X 0,Y 277.246,Z 269.006,A -85,B 0,C 180,E1 -17325.219,E2 -17325.219} C_VEL
LIN {X 0,Y 278.087,Z 273.505,A -85,B 0,C 180,E1 -17329.306,E2 -17329.306} C_VEL
LIN {X 0,Y 278.52,Z 275.988,A -85,B 0,C 180,E1 -17331.468,E2 -17331.468} C_VEL
LIN {X 0,Y 278.62,Z 279.688,A -85,B 0,C 180,E1 -17334.539,E2 -17334.539} C_VEL
LIN {X 0,Y 277.972,Z 284.005,A -85,B 0,C 180,E1 -17337.931,E2 -17337.931} C_VEL
LIN {X 0,Y 276.988,Z 290.395,A -85,B 0,C 180,E1 -17342.825,E2 -17342.825} C_VEL
LIN {X 0,Y 276.637,Z 293.857,A -85,B 0,C 180,E1 -17345.427,E2 -17345.427} C_VEL
LIN {X 0,Y 279.198,Z 307.438,A -85,B 0,C 180,E1 -17346.299,E2 -17346.299} C_VEL
LIN {X 0,Y 281.166,Z 320.847,A -85,B 0,C 180,E1 -17347.44,E2 -17347.44} C_VEL
LIN {X 0,Y 282.409,Z 332.312,A -85,B 0,C 180,E1 -17348.657,E2 -17348.657} C_VEL
LIN {X 0,Y 282.68,Z 340.162,A -85,B 0,C 180,E1 -17349.631,E2 -17349.631} C_VEL
LIN {X 0,Y 280.974,Z 351.515,A -85,B 0,C 180,E1 -17351.214,E2 -17351.214} C_VEL
LIN {X 0,Y 279.578,Z 361.385,A -85,B 0,C 180,E1 -17352.957,E2 -17352.957} C_VEL
LIN {X 0,Y 278.468,Z 369.171,A -85,B 0,C 180,E1 -17354.633,E2 -17354.633} C_VEL
LIN {X 0,Y 277.225,Z 377.418,A -85,B 0,C 180,E1 -17356.811,E2 -17356.811} C_VEL
LIN {X 0,Y 276.318,Z 384.058,A -85,B 0,C 180,E1 -17359.003,E2 -17359.003} C_VEL
LIN {X 0,Y 275.738,Z 389.339,A -85,B 0,C 180,E1 -17361.203,E2 -17361.203} C_VEL
LIN {X 0,Y 275.41,Z 393.421,A -85,B 0,C 180,E1 -17363.406,E2 -17363.406} C_VEL
LIN {X 0,Y 275.253,Z 396.419,A -85,B 0,C 180,E1 -17365.607,E2 -17365.607} C_VEL
LIN {X 0,Y 275.277,Z 397.868,A -85,B 0,C 180,E1 -17367.073,E2 -17367.073} C_VEL
LIN {X 0,Y 275.268,Z 398.874,A -85,B 0,C 180,E1 -17368.537,E2 -17368.537} C_VEL
LIN {X 0,Y 275.28,Z 399.483,A -85,B 0,C 180,E1 -17370,E2 -17370} C_VEL
LIN {X 0,Y 275.258,Z 399.697,A -85,B 0,C 180,E1 -17371.463,E2 -17371.463} C_VEL
LIN {X 0,Y 275.247,Z 399.487,A -85,B 0,C 180,E1 -17372.927,E2 -17372.927} C_VEL
LIN {X 0,Y 275.306,Z 397.848,A -85,B 0,C 180,E1 -17375.86,E2 -17375.86} C_VEL
LIN {X 0,Y 275.514,Z 396.441,A -85,B 0,C 180,E1 -17377.327,E2 -17377.327} C_VEL
LIN {X 0,Y 276.014,Z 393.503,A -85,B 0,C 180,E1 -17379.526,E2 -17379.526} C_VEL
LIN {X 0,Y 276.851,Z 389.552,A -85,B 0,C 180,E1 -17381.717,E2 -17381.717} C_VEL
LIN {X 0,Y 277.972,Z 384.498,A -85,B 0,C 180,E1 -17383.897,E2 -17383.897} C_VEL
LIN {X 0,Y 279.675,Z 378.212,A -85,B 0,C 180,E1 -17386.046,E2 -17386.046} C_VEL
LIN {X 0,Y 281.101,Z 371.971,A -85,B 0,C 180,E1 -17387.797,E2 -17387.797} C_VEL
LIN {X 0,Y 282.824,Z 364.258,A -85,B 0,C 180,E1 -17389.6,E2 -17389.6} C_VEL
LIN {X 0,Y 285.24,Z 354.08,A -85,B 0,C 180,E1 -17391.5,E2 -17391.5} C_VEL
LIN {X 0,Y 287.435,Z 343.836,A -85,B 0,C 180,E1 -17393.029,E2 -17393.029} C_VEL
LIN {X 0,Y 287.212,Z 333.033,A -85,B 0,C 180,E1 -17394.581,E2 -17394.581} C_VEL
LIN {X 0,Y 286.07,Z 322.519,A -85,B 0,C 180,E1 -17395.948,E2 -17395.948} C_VEL
LIN {X 0,Y 283.803,Z 311.278,A -85,B 0,C 180,E1 -17397.301,E2 -17397.301} C_VEL
LIN {X 0,Y 279.94,Z 298.502,A -85,B 0,C 180,E1 -17398.756,E2 -17398.756} C_VEL
LIN {X 0,Y 278.007,Z 292.928,A -85,B 0,C 180,E1 -17399.356,E2 -17399.356} C_VEL
LIN {X 0,Y 277.874,Z 292.176,A -85,B 0,C 180,E1 -17399.419,E2 -17399.419} C_VEL
LIN {X 0,Y 278.812,Z 287.188,A -85,B 0,C 180,E1 -17403.711,E2 -17403.711} C_VEL
LIN {X 0,Y 279.258,Z 283.485,A -85,B 0,C 180,E1 -17407.156,E2 -17407.156} C_VEL
LIN {X 0,Y 279.232,Z 281.664,A -85,B 0,C 180,E1 -17408.992,E2 -17408.992} C_VEL
LIN {X 0,Y 278.792,Z 278.169,A -85,B 0,C 180,E1 -17412.892,E2 -17412.892} C_VEL
LIN {X 0,Y 278.295,Z 274.922,A -85,B 0,C 180,E1 -17417.01,E2 -17417.01} C_VEL
LIN {X 0,Y 277.862,Z 272.383,A -85,B 0,C 180,E1 -17420.776,E2 -17420.776} C_VEL
LIN {X 0,Y 277.532,Z 270.334,A -85,B 0,C 180,E1 -17424.376,E2 -17424.376} C_VEL
LIN {X 0,Y 277.244,Z 268.951,A -85,B 0,C 180,E1 -17427.835,E2 -17427.835} C_VEL
LIN {X 0,Y 277.288,Z 268.944,A -85,B 0,C 180,E1 -17431.211,E2 -17431.211} C_VEL
LIN {X 0,Y 277.312,Z 268.943,A -85,B 0,C 180,E1 -17434.478,E2 -17434.478} C_VEL
LIN {X 0,Y 277.282,Z 268.946,A -85,B 0,C 180,E1 -17437.653,E2 -17437.653} C_VEL
LIN {X 0,Y 277.342,Z 268.94,A -85,B 0,C 180,E1 -17440.764,E2 -17440.764} C_VEL
LIN {X 0,Y 277.424,Z 268.928,A -85,B 0,C 180,E1 -17445.324,E2 -17445.324} C_VEL
LIN {X 0,Y 277.502,Z 268.919,A -85,B 0,C 180,E1 -17449.787,E2 -17449.787} C_VEL
LIN {X 0,Y 277.648,Z 268.902,A -85,B 0,C 180,E1 -17452.727,E2 -17452.727} C_VEL
LIN {X 0,Y 277.72,Z 269.177,A -85,B 0,C 180,E1 -17457.097,E2 -17457.097} C_VEL
LIN {X 0,Y 278.134,Z 270.421,A -85,B 0,C 180,E1 -17459.998,E2 -17459.998} C_VEL
LIN {X 0,Y 278.148,Z 271.93,A -85,B 0,C 180,E1 -17462.895,E2 -17462.895} C_VEL
LIN {X 0,Y 278.323,Z 274.495,A -85,B 0,C 180,E1 -17467.251,E2 -17467.251} C_VEL
LIN {X 0,Y 278.299,Z 276.44,A -85,B 0,C 180,E1 -17470.18,E2 -17470.18} C_VEL
LIN {X 0,Y 277.707,Z 279.796,A -85,B 0,C 180,E1 -17474.657,E2 -17474.657} C_VEL
LIN {X 0,Y 277.435,Z 281.337,A -85,B 0,C 180,E1 -17476.603,E2 -17476.603} C_VEL
LIN {X 0,Y 278.499,Z 284.479,A -85,B 0,C 180,E1 -17476.946,E2 -17476.946} C_VEL
LIN {X 0,Y 281.861,Z 292.418,A -85,B 0,C 180,E1 -17477.971,E2 -17477.971} C_VEL
LIN {X 0,Y 285.486,Z 303.581,A -85,B 0,C 180,E1 -17479.409,E2 -17479.409} C_VEL
LIN {X 0,Y 287.796,Z 313.338,A -85,B 0,C 180,E1 -17480.736,E2 -17480.736} C_VEL
LIN {X 0,Y 289.249,Z 323.378,A -85,B 0,C 180,E1 -17482.197,E2 -17482.197} C_VEL
LIN {X 0,Y 289.141,Z 326.916,A -85,B 0,C 180,E1 -17482.697,E2 -17482.697} C_VEL
LIN {X 0,Y 287.047,Z 337.544,A -85,B 0,C 180,E1 -17484.209,E2 -17484.209} C_VEL
LIN {X 0,Y 284.782,Z 347.446,A -85,B 0,C 180,E1 -17485.977,E2 -17485.977} C_VEL
LIN {X 0,Y 282.697,Z 355.948,A -85,B 0,C 180,E1 -17487.861,E2 -17487.861} C_VEL
LIN {X 0,Y 280.655,Z 363.881,A -85,B 0,C 180,E1 -17490.053,E2 -17490.053} C_VEL
LIN {X 0,Y 278.912,Z 370.292,A -85,B 0,C 180,E1 -17492.313,E2 -17492.313} C_VEL
LIN {X 0,Y 277.523,Z 375.599,A -85,B 0,C 180,E1 -17494.733,E2 -17494.733} C_VEL
LIN {X 0,Y 276.348,Z 380.178,A -85,B 0,C 180,E1 -17497.613,E2 -17497.613} C_VEL
LIN {X 0,Y 275.581,Z 382.719,A -85,B 0,C 180,E1 -17500.088,E2 -17500.088} C_VEL
LIN {X 0,Y 275.209,Z 383.985,A -85,B 0,C 180,E1 -17502.222,E2 -17502.222} C_VEL
LIN {X 0,Y 274.971,Z 384.388,A -85,B 0,C 180,E1 -17504.305,E2 -17504.305} C_VEL
LIN {X 0,Y 274.91,Z 383.987,A -85,B 0,C 180,E1 -17506.352,E2 -17506.352} C_VEL
LIN {X 0,Y 274.938,Z 382.86,A -85,B 0,C 180,E1 -17508.348,E2 -17508.348} C_VEL
LIN {X 0,Y 275.163,Z 381.015,A -85,B 0,C 180,E1 -17510.319,E2 -17510.319} C_VEL
LIN {X 0,Y 275.55,Z 378.398,A -85,B 0,C 180,E1 -17512.258,E2 -17512.258} C_VEL
LIN {X 0,Y 276.09,Z 374.292,A -85,B 0,C 180,E1 -17514.541,E2 -17514.541} C_VEL
LIN {X 0,Y 276.823,Z 368.717,A -85,B 0,C 180,E1 -17516.905,E2 -17516.905} C_VEL
LIN {X 0,Y 277.882,Z 361.403,A -85,B 0,C 180,E1 -17519.302,E2 -17519.302} C_VEL
LIN {X 0,Y 279.147,Z 353.277,A -85,B 0,C 180,E1 -17521.423,E2 -17521.423} C_VEL
LIN {X 0,Y 280.567,Z 343.586,A -85,B 0,C 180,E1 -17523.445,E2 -17523.445} C_VEL
LIN {X 0,Y 282.006,Z 333.509,A -85,B 0,C 180,E1 -17525.132,E2 -17525.132} C_VEL
LIN {X 0,Y 283.478,Z 322.361,A -85,B 0,C 180,E1 -17526.63,E2 -17526.63} C_VEL
LIN {X 0,Y 283.932,Z 318.606,A -85,B 0,C 180,E1 -17527.056,E2 -17527.056} C_VEL
LIN {X 0,Y 282.4,Z 307.938,A -85,B 0,C 180,E1 -17528.274,E2 -17528.274} C_VEL
LIN {X 0,Y 279.945,Z 295.282,A -85,B 0,C 180,E1 -17529.464,E2 -17529.464} C_VEL
LIN {X 0,Y 276.642,Z 281.552,A -85,B 0,C 180,E1 -17530.484,E2 -17530.484} C_VEL
LIN {X 0,Y 276.256,Z 279.563,A -85,B 0,C 180,E1 -17530.63,E2 -17530.63} C_VEL
LIN {X 0,Y 276.689,Z 274.973,A -85,B 0,C 180,E1 -17535.286,E2 -17535.286} C_VEL
LIN {X 0,Y 277.117,Z 270.701,A -85,B 0,C 180,E1 -17539.775,E2 -17539.775} C_VEL
LIN {X 0,Y 277.417,Z 268.929,A -85,B 0,C 180,E1 -17541.794,E2 -17541.794} C_VEL
LIN {X 0,Y 277.518,Z 268.914,A -85,B 0,C 180,E1 -17544.186,E2 -17544.186} C_VEL
LIN {X 0,Y 277.813,Z 268.881,A -85,B 0,C 180,E1 -17548.551,E2 -17548.551} C_VEL
LIN {X 0,Y 277.815,Z 268.877,A -85,B 0,C 180,E1 -17551.45,E2 -17551.45} C_VEL
LIN {X 0,Y 277.643,Z 268.899,A -85,B 0,C 180,E1 -17557.271,E2 -17557.271} C_VEL
LIN {X 0,Y 277.497,Z 268.92,A -85,B 0,C 180,E1 -17560.212,E2 -17560.212} C_VEL
LIN {X 0,Y 277.425,Z 268.927,A -85,B 0,C 180,E1 -17564.675,E2 -17564.675} C_VEL
LIN {X 0,Y 277.337,Z 268.935,A -85,B 0,C 180,E1 -17569.234,E2 -17569.234} C_VEL
LIN {X 0,Y 277.334,Z 268.941,A -85,B 0,C 180,E1 -17573.92,E2 -17573.92} C_VEL
LIN {X 0,Y 277.316,Z 268.938,A -85,B 0,C 180,E1 -17577.506,E2 -17577.506} C_VEL
LIN {X 0,Y 277.262,Z 268.944,A -85,B 0,C 180,E1 -17580.482,E2 -17580.482} C_VEL
LIN {X 0,Y 277.245,Z 268.951,A -85,B 0,C 180,E1 -17583.895,E2 -17583.895} C_VEL
LIN {X 0,Y 277.282,Z 268.946,A -85,B 0,C 180,E1 -17587.466,E2 -17587.466} C_VEL
LIN {X 0,Y 277.285,Z 268.94,A -85,B 0,C 180,E1 -17591.222,E2 -17591.222} C_VEL
LIN {X 0,Y 277.279,Z 268.943,A -85,B 0,C 180,E1 -17595.209,E2 -17595.209} C_VEL
LIN {X 0,Y 277.287,Z 268.946,A -85,B 0,C 180,E1 -17599.496,E2 -17599.496} C_VEL
LIN {X 0,Y 277.278,Z 268.944,A -85,B 0,C 180,E1 -17602.535,E2 -17602.535} C_VEL
LIN {X 0,Y 277.246,Z 268.943,A -85,B 0,C 180,E1 -17606.107,E2 -17606.107} C_VEL
LIN {X 0,Y 277.254,Z 268.94,A -85,B 0,C 180,E1 -17609.54,E2 -17609.54} C_VEL
LIN {X 0,Y 277.352,Z 268.934,A -85,B 0,C 180,E1 -17612.866,E2 -17612.866} C_VEL
LIN {X 0,Y 277.321,Z 268.938,A -85,B 0,C 180,E1 -17616.081,E2 -17616.081} C_VEL
LIN {X 0,Y 277.338,Z 268.94,A -85,B 0,C 180,E1 -17620.768,E2 -17620.768} C_VEL
LIN {X 0,Y 277.422,Z 268.92,A -85,B 0,C 180,E1 -17625.327,E2 -17625.327} C_VEL
LIN {X 0,Y 277.456,Z 268.915,A -85,B 0,C 180,E1 -17629.789,E2 -17629.789} C_VEL
LIN {X 0,Y 277.635,Z 268.9,A -85,B 0,C 180,E1 -17632.73,E2 -17632.73} C_VEL
LIN {X 0,Y 277.817,Z 268.878,A -85,B 0,C 180,E1 -17638.552,E2 -17638.552} C_VEL
LIN {X 0,Y 277.818,Z 268.874,A -85,B 0,C 180,E1 -17641.451,E2 -17641.451} C_VEL
LIN {X 0,Y 277.65,Z 268.894,A -85,B 0,C 180,E1 -17647.273,E2 -17647.273} C_VEL
LIN {X 0,Y 277.505,Z 268.918,A -85,B 0,C 180,E1 -17650.213,E2 -17650.213} C_VEL
LIN {X 0,Y 277.435,Z 268.924,A -85,B 0,C 180,E1 -17651.276,E2 -17651.276} C_VEL
LIN {X 0,Y 276.747,Z 269.013,A -85,B 0,C 180,E1 -17652.488,E2 -17652.488} C_VEL
LIN {X 0,Y 273.853,Z 269.37,A -85,B 0,C 180,E1 -17654.462,E2 -17654.462} C_VEL
LIN {X 0,Y 271.407,Z 269.675,A -85,B 0,C 180,E1 -17656.067,E2 -17656.067} C_VEL
LIN {X 0,Y 270.363,Z 269.803,A -85,B 0,C 180,E1 -17657.311,E2 -17657.311} C_VEL
LIN {X 0,Y 270.28,Z 269.81,A -85,B 0,C 180,E1 -17657.733,E2 -17657.733} C_VEL
LIN {X 0,Y 270.221,Z 269.823,A -85,B 0,C 180,E1 -17661.355,E2 -17661.355} C_VEL
LIN {X 0,Y 270.274,Z 269.816,A -85,B 0,C 180,E1 -17664.587,E2 -17664.587} C_VEL
LIN {X 0,Y 270.27,Z 269.816,A -85,B 0,C 180,E1 -17667.91,E2 -17667.91} C_VEL
LIN {X 0,Y 270.185,Z 269.832,A -85,B 0,C 180,E1 -17671.35,E2 -17671.35} C_VEL
LIN {X 0,Y 270.203,Z 269.827,A -85,B 0,C 180,E1 -17674.907,E2 -17674.907} C_VEL
LIN {X 0,Y 270.2,Z 269.827,A -85,B 0,C 180,E1 -17678.712,E2 -17678.712} C_VEL
LIN {X 0,Y 270.174,Z 269.83,A -85,B 0,C 180,E1 -17682.56,E2 -17682.56} C_VEL
LIN {X 0,Y 270.202,Z 269.907,A -85,B 0,C 180,E1 -17685.013,E2 -17685.013} C_VEL
LIN {X 0,Y 270.957,Z 273.942,A -85,B 0,C 180,E1 -17688.783,E2 -17688.783} C_VEL
LIN {X 0,Y 271.484,Z 277.074,A -85,B 0,C 180,E1 -17691.59,E2 -17691.59} C_VEL
LIN {X 0,Y 271.584,Z 280.369,A -85,B 0,C 180,E1 -17694.392,E2 -17694.392} C_VEL
LIN {X 0,Y 270.92,Z 284.68,A -85,B 0,C 180,E1 -17697.874,E2 -17697.874} C_VEL
LIN {X 0,Y 269.986,Z 290.261,A -85,B 0,C 180,E1 -17702.261,E2 -17702.261} C_VEL
LIN {X 0,Y 269.619,Z 293.681,A -85,B 0,C 180,E1 -17704.904,E2 -17704.904} C_VEL
LIN {X 0,Y 272.196,Z 307.18,A -85,B 0,C 180,E1 -17705.807,E2 -17705.807} C_VEL
LIN {X 0,Y 274.097,Z 320.505,A -85,B 0,C 180,E1 -17706.972,E2 -17706.972} C_VEL
LIN {X 0,Y 275.449,Z 332.578,A -85,B 0,C 180,E1 -17708.295,E2 -17708.295} C_VEL
LIN {X 0,Y 275.783,Z 340.327,A -85,B 0,C 180,E1 -17709.293,E2 -17709.293} C_VEL
LIN {X 0,Y 274.041,Z 351.608,A -85,B 0,C 180,E1 -17710.914,E2 -17710.914} C_VEL
LIN {X 0,Y 272.57,Z 361.52,A -85,B 0,C 180,E1 -17712.722,E2 -17712.722} C_VEL
LIN {X 0,Y 271.333,Z 369.905,A -85,B 0,C 180,E1 -17714.604,E2 -17714.604} C_VEL
LIN {X 0,Y 270.059,Z 377.988,A -85,B 0,C 180,E1 -17716.838,E2 -17716.838} C_VEL
LIN {X 0,Y 269.319,Z 383.474,A -85,B 0,C 180,E1 -17718.713,E2 -17718.713} C_VEL
LIN {X 0,Y 268.699,Z 388.83,A -85,B 0,C 180,E1 -17720.971,E2 -17720.971} C_VEL
LIN {X 0,Y 268.334,Z 392.982,A -85,B 0,C 180,E1 -17723.231,E2 -17723.231} C_VEL
LIN {X 0,Y 268.166,Z 396.048,A -85,B 0,C 180,E1 -17725.49,E2 -17725.49} C_VEL
LIN {X 0,Y 268.187,Z 397.556,A -85,B 0,C 180,E1 -17726.996,E2 -17726.996} C_VEL
LIN {X 0,Y 268.194,Z 398.597,A -85,B 0,C 180,E1 -17728.498,E2 -17728.498} C_VEL
LIN {X 0,Y 268.204,Z 399.236,A -85,B 0,C 180,E1 -17730,E2 -17730} C_VEL
LIN {X 0,Y 268.184,Z 399.479,A -85,B 0,C 180,E1 -17731.501,E2 -17731.501} C_VEL
LIN {X 0,Y 268.158,Z 399.322,A -85,B 0,C 180,E1 -17733.004,E2 -17733.004} C_VEL
LIN {X 0,Y 268.231,Z 397.745,A -85,B 0,C 180,E1 -17736.016,E2 -17736.016} C_VEL
LIN {X 0,Y 268.455,Z 396.368,A -85,B 0,C 180,E1 -17737.521,E2 -17737.521} C_VEL
LIN {X 0,Y 268.991,Z 393.496,A -85,B 0,C 180,E1 -17739.777,E2 -17739.777} C_VEL
LIN {X 0,Y 269.875,Z 389.627,A -85,B 0,C 180,E1 -17742.024,E2 -17742.024} C_VEL
LIN {X 0,Y 271.077,Z 384.665,A -85,B 0,C 180,E1 -17744.258,E2 -17744.258} C_VEL
LIN {X 0,Y 272.876,Z 378.463,A -85,B 0,C 180,E1 -17746.457,E2 -17746.457} C_VEL
LIN {X 0,Y 274.475,Z 371.501,A -85,B 0,C 180,E1 -17748.477,E2 -17748.477} C_VEL
LIN {X 0,Y 276.599,Z 363.067,A -85,B 0,C 180,E1 -17750.448,E2 -17750.448} C_VEL
LIN {X 0,Y 279.209,Z 352.652,A -85,B 0,C 180,E1 -17752.377,E2 -17752.377} C_VEL
LIN {X 0,Y 280.943,Z 344.729,A -85,B 0,C 180,E1 -17753.593,E2 -17753.593} C_VEL
LIN {X 0,Y 280.792,Z 334.266,A -85,B 0,C 180,E1 -17755.181,E2 -17755.181} C_VEL
LIN {X 0,Y 279.714,Z 323.575,A -85,B 0,C 180,E1 -17756.642,E2 -17756.642} C_VEL
LIN {X 0,Y 277.166,Z 311.267,A -85,B 0,C 180,E1 -17758.227,E2 -17758.227} C_VEL
LIN {X 0,Y 273.564,Z 299.235,A -85,B 0,C 180,E1 -17759.695,E2 -17759.695} C_VEL
LIN {X 0,Y 271.172,Z 292.555,A -85,B 0,C 180,E1 -17760.465,E2 -17760.465} C_VEL
LIN {X 0,Y 271.087,Z 291.898,A -85,B 0,C 180,E1 -17760.55,E2 -17760.55} C_VEL
LIN {X 0,Y 271.938,Z 287.346,A -85,B 0,C 180,E1 -17764.65,E2 -17764.65} C_VEL
LIN {X 0,Y 272.247,Z 285.068,A -85,B 0,C 180,E1 -17766.843,E2 -17766.843} C_VEL
LIN {X 0,Y 272.111,Z 281.88,A -85,B 0,C 180,E1 -17770.216,E2 -17770.216} C_VEL
LIN {X 0,Y 271.657,Z 278.449,A -85,B 0,C 180,E1 -17774.306,E2 -17774.306} C_VEL
LIN {X 0,Y 271.165,Z 275.26,A -85,B 0,C 180,E1 -17778.729,E2 -17778.729} C_VEL
LIN {X 0,Y 270.872,Z 273.544,A -85,B 0,C 180,E1 -17781.485,E2 -17781.485} C_VEL
LIN {X 0,Y 270.524,Z 271.595,A -85,B 0,C 180,E1 -17785.14,E2 -17785.14} C_VEL
LIN {X 0,Y 270.223,Z 269.919,A -85,B 0,C 180,E1 -17789.121,E2 -17789.121} C_VEL
LIN {X 0,Y 270.264,Z 269.819,A -85,B 0,C 180,E1 -17792.144,E2 -17792.144} C_VEL
LIN {X 0,Y 270.275,Z 269.82,A -85,B 0,C 180,E1 -17795.517,E2 -17795.517} C_VEL
LIN {X 0,Y 270.299,Z 269.816,A -85,B 0,C 180,E1 -17800.243,E2 -17800.243} C_VEL
LIN {X 0,Y 270.393,Z 269.805,A -85,B 0,C 180,E1 -17804.933,E2 -17804.933} C_VEL
LIN {X 0,Y 270.437,Z 269.8,A -85,B 0,C 180,E1 -17809.517,E2 -17809.517} C_VEL
LIN {X 0,Y 270.606,Z 269.778,A -85,B 0,C 180,E1 -17812.537,E2 -17812.537} C_VEL
LIN {X 0,Y 270.538,Z 269.787,A -85,B 0,C 180,E1 -17814.034,E2 -17814.034} C_VEL
LIN {X 0,Y 271.001,Z 271.267,A -85,B 0,C 180,E1 -17818.512,E2 -17818.512} C_VEL
LIN {X 0,Y 271.212,Z 271.895,A -85,B 0,C 180,E1 -17819.998,E2 -17819.998} C_VEL
LIN {X 0,Y 271.188,Z 273.402,A -85,B 0,C 180,E1 -17822.969,E2 -17822.969} C_VEL
LIN {X 0,Y 271.344,Z 275.955,A -85,B 0,C 180,E1 -17827.439,E2 -17827.439} C_VEL
LIN {X 0,Y 271.268,Z 277.919,A -85,B 0,C 180,E1 -17830.447,E2 -17830.447} C_VEL
LIN {X 0,Y 270.65,Z 281.281,A -85,B 0,C 180,E1 -17835.049,E2 -17835.049} C_VEL
LIN {X 0,Y 270.635,Z 281.834,A -85,B 0,C 180,E1 -17835.511,E2 -17835.511} C_VEL
LIN {X 0,Y 271.868,Z 285.103,A -85,B 0,C 180,E1 -17835.915,E2 -17835.915} C_VEL
LIN {X 0,Y 276.295,Z 295.797,A -85,B 0,C 180,E1 -17837.388,E2 -17837.388} C_VEL
LIN {X 0,Y 279.88,Z 307.689,A -85,B 0,C 180,E1 -17839.051,E2 -17839.051} C_VEL
LIN {X 0,Y 281.851,Z 317.174,A -85,B 0,C 180,E1 -17840.43,E2 -17840.43} C_VEL
LIN {X 0,Y 282.996,Z 326.392,A -85,B 0,C 180,E1 -17841.869,E2 -17841.869} C_VEL
LIN {X 0,Y 281.038,Z 336.511,A -85,B 0,C 180,E1 -17843.327,E2 -17843.327} C_VEL
LIN {X 0,Y 278.689,Z 346.467,A -85,B 0,C 180,E1 -17845.089,E2 -17845.089} C_VEL
LIN {X 0,Y 276.163,Z 356.18,A -85,B 0,C 180,E1 -17847.261,E2 -17847.261} C_VEL
LIN {X 0,Y 274.147,Z 363.641,A -85,B 0,C 180,E1 -17849.355,E2 -17849.355} C_VEL
LIN {X 0,Y 272.296,Z 370.017,A -85,B 0,C 180,E1 -17851.601,E2 -17851.601} C_VEL
LIN {X 0,Y 270.898,Z 375.062,A -85,B 0,C 180,E1 -17853.884,E2 -17853.884} C_VEL
LIN {X 0,Y 269.789,Z 378.902,A -85,B 0,C 180,E1 -17856.145,E2 -17856.145} C_VEL
LIN {X 0,Y 268.834,Z 382.126,A -85,B 0,C 180,E1 -17858.857,E2 -17858.857} C_VEL
LIN {X 0,Y 268.321,Z 383.674,A -85,B 0,C 180,E1 -17860.903,E2 -17860.903} C_VEL
LIN {X 0,Y 268.012,Z 384.485,A -85,B 0,C 180,E1 -17862.981,E2 -17862.981} C_VEL
LIN {X 0,Y 267.845,Z 384.497,A -85,B 0,C 180,E1 -17865.106,E2 -17865.106} C_VEL
LIN {X 0,Y 267.802,Z 383.696,A -85,B 0,C 180,E1 -17867.288,E2 -17867.288} C_VEL
LIN {X 0,Y 267.937,Z 381.999,A -85,B 0,C 180,E1 -17869.52,E2 -17869.52} C_VEL
LIN {X 0,Y 268.331,Z 379.318,A -85,B 0,C 180,E1 -17871.786,E2 -17871.786} C_VEL
LIN {X 0,Y 268.869,Z 375.464,A -85,B 0,C 180,E1 -17874.123,E2 -17874.123} C_VEL
LIN {X 0,Y 269.709,Z 369.485,A -85,B 0,C 180,E1 -17876.825,E2 -17876.825} C_VEL
LIN {X 0,Y 270.799,Z 362.075,A -85,B 0,C 180,E1 -17879.365,E2 -17879.365} C_VEL
LIN {X 0,Y 272.034,Z 354.43,A -85,B 0,C 180,E1 -17881.444,E2 -17881.444} C_VEL
LIN {X 0,Y 273.422,Z 345.462,A -85,B 0,C 180,E1 -17883.427,E2 -17883.427} C_VEL
LIN {X 0,Y 274.897,Z 335.182,A -85,B 0,C 180,E1 -17885.252,E2 -17885.252} C_VEL
LIN {X 0,Y 276.47,Z 324.119,A -85,B 0,C 180,E1 -17886.814,E2 -17886.814} C_VEL
LIN {X 0,Y 276.99,Z 318.958,A -85,B 0,C 180,E1 -17887.438,E2 -17887.438} C_VEL
LIN {X 0,Y 275.405,Z 308.128,A -85,B 0,C 180,E1 -17888.716,E2 -17888.716} C_VEL
LIN {X 0,Y 272.912,Z 295.429,A -85,B 0,C 180,E1 -17889.951,E2 -17889.951} C_VEL
LIN {X 0,Y 269.676,Z 281.955,A -85,B 0,C 180,E1 -17890.989,E2 -17890.989} C_VEL
LIN {X 0,Y 269.208,Z 279.74,A -85,B 0,C 180,E1 -17891.152,E2 -17891.152} C_VEL
LIN {X 0,Y 269.602,Z 276.139,A -85,B 0,C 180,E1 -17894.89,E2 -17894.89} C_VEL
LIN {X 0,Y 270.017,Z 271.823,A -85,B 0,C 180,E1 -17899.503,E2 -17899.503} C_VEL
LIN {X 0,Y 270.395,Z 269.804,A -85,B 0,C 180,E1 -17901.842,E2 -17901.842} C_VEL
LIN {X 0,Y 270.483,Z 269.789,A -85,B 0,C 180,E1 -17904.035,E2 -17904.035} C_VEL
LIN {X 0,Y 270.778,Z 269.757,A -85,B 0,C 180,E1 -17908.513,E2 -17908.513} C_VEL
LIN {X 0,Y 270.781,Z 269.753,A -85,B 0,C 180,E1 -17911.487,E2 -17911.487} C_VEL
LIN {X 0,Y 270.601,Z 269.776,A -85,B 0,C 180,E1 -17917.462,E2 -17917.462} C_VEL
LIN {X 0,Y 270.432,Z 269.798,A -85,B 0,C 180,E1 -17920.481,E2 -17920.481} C_VEL
LIN {X 0,Y 270.393,Z 269.801,A -85,B 0,C 180,E1 -17925.065,E2 -17925.065} C_VEL
LIN {X 0,Y 270.294,Z 269.814,A -85,B 0,C 180,E1 -17929.756,E2 -17929.756} C_VEL
LIN {X 0,Y 270.269,Z 269.816,A -85,B 0,C 180,E1 -17934.586,E2 -17934.586} C_VEL
LIN {X 0,Y 270.261,Z 269.816,A -85,B 0,C 180,E1 -17937.909,E2 -17937.909} C_VEL
LIN {X 0,Y 270.176,Z 269.828,A -85,B 0,C 180,E1 -17941.349,E2 -17941.349} C_VEL
LIN {X 0,Y 270.207,Z 269.825,A -85,B 0,C 180,E1 -17944.904,E2 -17944.904} C_VEL
LIN {X 0,Y 270.213,Z 269.821,A -85,B 0,C 180,E1 -17948.718,E2 -17948.718} C_VEL
LIN {X 0,Y 270.248,Z 269.812,A -85,B 0,C 180,E1 -17952.543,E2 -17952.543} C_VEL
LIN {X 0,Y 270.223,Z 269.821,A -85,B 0,C 180,E1 -17956.737,E2 -17956.737} C_VEL
LIN {X 0,Y 270.24,Z 269.824,A -85,B 0,C 180,E1 -17959.449,E2 -17959.449} C_VEL
LIN {X 0,Y 270.248,Z 269.818,A -85,B 0,C 180,E1 -17963.723,E2 -17963.723} C_VEL
LIN {X 0,Y 270.196,Z 269.824,A -85,B 0,C 180,E1 -17966.894,E2 -17966.894} C_VEL
LIN {X 0,Y 270.221,Z 269.814,A -85,B 0,C 180,E1 -17970.388,E2 -17970.388} C_VEL
LIN {X 0,Y 270.256,Z 269.816,A -85,B 0,C 180,E1 -17973.765,E2 -17973.765} C_VEL
LIN {X 0,Y 270.226,Z 269.825,A -85,B 0,C 180,E1 -17977.04,E2 -17977.04} C_VEL
LIN {X 0,Y 270.295,Z 269.814,A -85,B 0,C 180,E1 -17980.246,E2 -17980.246} C_VEL
LIN {X 0,Y 270.39,Z 269.797,A -85,B 0,C 180,E1 -17984.937,E2 -17984.937} C_VEL
LIN {X 0,Y 270.408,Z 269.792,A -85,B 0,C 180,E1 -17989.52,E2 -17989.52} C_VEL
LIN {X 0,Y 270.594,Z 269.778,A -85,B 0,C 180,E1 -17992.54,E2 -17992.54} C_VEL
LIN {X 0,Y 270.783,Z 269.755,A -85,B 0,C 180,E1 -17998.515,E2 -17998.515} C_VEL
LIN {X 0,Y 270.784,Z 269.75,A -85,B 0,C 180,E1 -18001.489,E2 -18001.489} C_VEL
LIN {X 0,Y 270.608,Z 269.771,A -85,B 0,C 180,E1 -18007.463,E2 -18007.463} C_VEL
LIN {X 0,Y 270.44,Z 269.796,A -85,B 0,C 180,E1 -18010.483,E2 -18010.483} C_VEL
LIN {X 0,Y 270.395,Z 269.8,A -85,B 0,C 180,E1 -18015.067,E2 -18015.067} C_VEL
LIN {X 0,Y 270.28,Z 269.81,A -85,B 0,C 180,E1 -18017.733,E2 -18017.733} C_VEL
LIN {X 0,Y 269.605,Z 269.898,A -85,B 0,C 180,E1 -18018.976,E2 -18018.976} C_VEL
LIN {X 0,Y 266.709,Z 270.264,A -85,B 0,C 180,E1 -18021.002,E2 -18021.002} C_VEL
LIN {X 0,Y 264.272,Z 270.567,A -85,B 0,C 180,E1 -18022.649,E2 -18022.649} C_VEL
LIN {X 0,Y 263.261,Z 270.692,A -85,B 0,C 180,E1 -18023.926,E2 -18023.926} C_VEL
LIN {X 0,Y 263.197,Z 270.698,A -85,B 0,C 180,E1 -18024.359,E2 -18024.359} C_VEL
LIN {X 0,Y 263.176,Z 270.698,A -85,B 0,C 180,E1 -18028.732,E2 -18028.732} C_VEL
LIN {X 0,Y 263.134,Z 270.707,A -85,B 0,C 180,E1 -18032.29,E2 -18032.29} C_VEL
LIN {X 0,Y 263.185,Z 270.7,A -85,B 0,C 180,E1 -18036.765,E2 -18036.765} C_VEL
LIN {X 0,Y 263.127,Z 270.709,A -85,B 0,C 180,E1 -18041.595,E2 -18041.595} C_VEL
LIN {X 0,Y 263.178,Z 270.773,A -85,B 0,C 180,E1 -18044.777,E2 -18044.777} C_VEL
LIN {X 0,Y 264.052,Z 275.501,A -85,B 0,C 180,E1 -18049.301,E2 -18049.301} C_VEL
LIN {X 0,Y 264.507,Z 278.838,A -85,B 0,C 180,E1 -18052.331,E2 -18052.331} C_VEL
LIN {X 0,Y 264.545,Z 281.037,A -85,B 0,C 180,E1 -18054.236,E2 -18054.236} C_VEL
LIN {X 0,Y 264.012,Z 284.274,A -85,B 0,C 180,E1 -18056.927,E2 -18056.927} C_VEL
LIN {X 0,Y 263.086,Z 289.602,A -85,B 0,C 180,E1 -18061.26,E2 -18061.26} C_VEL
LIN {X 0,Y 262.625,Z 293.618,A -85,B 0,C 180,E1 -18064.37,E2 -18064.37} C_VEL
LIN {X 0,Y 265.132,Z 306.931,A -85,B 0,C 180,E1 -18065.283,E2 -18065.283} C_VEL
LIN {X 0,Y 267.055,Z 319.992,A -85,B 0,C 180,E1 -18066.464,E2 -18066.464} C_VEL
LIN {X 0,Y 268.394,Z 331.93,A -85,B 0,C 180,E1 -18067.805,E2 -18067.805} C_VEL
LIN {X 0,Y 268.866,Z 340.447,A -85,B 0,C 180,E1 -18068.936,E2 -18068.936} C_VEL
LIN {X 0,Y 267.117,Z 351.668,A -85,B 0,C 180,E1 -18070.6,E2 -18070.6} C_VEL
LIN {X 0,Y 265.567,Z 361.641,A -85,B 0,C 180,E1 -18072.477,E2 -18072.477} C_VEL
LIN {X 0,Y 264.45,Z 369.132,A -85,B 0,C 180,E1 -18074.193,E2 -18074.193} C_VEL
LIN {X 0,Y 263.132,Z 377.315,A -85,B 0,C 180,E1 -18076.485,E2 -18076.485} C_VEL
LIN {X 0,Y 262.314,Z 382.884,A -85,B 0,C 180,E1 -18078.408,E2 -18078.408} C_VEL
LIN {X 0,Y 261.674,Z 388.32,A -85,B 0,C 180,E1 -18080.726,E2 -18080.726} C_VEL
LIN {X 0,Y 261.259,Z 392.543,A -85,B 0,C 180,E1 -18083.047,E2 -18083.047} C_VEL
LIN {X 0,Y 261.072,Z 395.676,A -85,B 0,C 180,E1 -18085.368,E2 -18085.368} C_VEL
LIN {X 0,Y 261.1,Z 397.226,A -85,B 0,C 180,E1 -18086.914,E2 -18086.914} C_VEL
LIN {X 0,Y 261.122,Z 398.32,A -85,B 0,C 180,E1 -18088.458,E2 -18088.458} C_VEL
LIN {X 0,Y 261.129,Z 398.988,A -85,B 0,C 180,E1 -18090,E2 -18090} C_VEL
LIN {X 0,Y 261.111,Z 399.261,A -85,B 0,C 180,E1 -18091.542,E2 -18091.542} C_VEL
LIN {X 0,Y 261.054,Z 399.141,A -85,B 0,C 180,E1 -18093.086,E2 -18093.086} C_VEL
LIN {X 0,Y 261.09,Z 398.324,A -85,B 0,C 180,E1 -18095.137,E2 -18095.137} C_VEL
LIN {X 0,Y 261.385,Z 396.312,A -85,B 0,C 180,E1 -18097.726,E2 -18097.726} C_VEL
LIN {X 0,Y 261.987,Z 393.514,A -85,B 0,C 180,E1 -18100.041,E2 -18100.041} C_VEL
LIN {X 0,Y 262.916,Z 389.718,A -85,B 0,C 180,E1 -18102.347,E2 -18102.347} C_VEL
LIN {X 0,Y 264.199,Z 384.832,A -85,B 0,C 180,E1 -18104.637,E2 -18104.637} C_VEL
LIN {X 0,Y 266.43,Z 377.587,A -85,B 0,C 180,E1 -18107.262,E2 -18107.262} C_VEL
LIN {X 0,Y 268.267,Z 370.147,A -85,B 0,C 180,E1 -18109.414,E2 -18109.414} C_VEL
LIN {X 0,Y 270.448,Z 361.909,A -85,B 0,C 180,E1 -18111.334,E2 -18111.334} C_VEL
LIN {X 0,Y 273.274,Z 351.337,A -85,B 0,C 180,E1 -18113.291,E2 -18113.291} C_VEL
LIN {X 0,Y 274.489,Z 345.703,A -85,B 0,C 180,E1 -18114.183,E2 -18114.183} C_VEL
LIN {X 0,Y 274.352,Z 333.98,A -85,B 0,C 180,E1 -18116.03,E2 -18116.03} C_VEL
LIN {X 0,Y 273.213,Z 323.178,A -85,B 0,C 180,E1 -18117.582,E2 -18117.582} C_VEL
LIN {X 0,Y 270.844,Z 311.927,A -85,B 0,C 180,E1 -18119.117,E2 -18119.117} C_VEL
LIN {X 0,Y 267.176,Z 299.73,A -85,B 0,C 180,E1 -18120.712,E2 -18120.712} C_VEL
LIN {X 0,Y 265.265,Z 294.918,A -85,B 0,C 180,E1 -18121.361,E2 -18121.361} C_VEL
LIN {X 0,Y 264.292,Z 291.665,A -85,B 0,C 180,E1 -18121.735,E2 -18121.735} C_VEL
LIN {X 0,Y 265.078,Z 287.495,A -85,B 0,C 180,E1 -18125.681,E2 -18125.681} C_VEL
LIN {X 0,Y 265.248,Z 285.657,A -85,B 0,C 180,E1 -18127.545,E2 -18127.545} C_VEL
LIN {X 0,Y 265.176,Z 283.623,A -85,B 0,C 180,E1 -18129.77,E2 -18129.77} C_VEL
LIN {X 0,Y 264.795,Z 280.416,A -85,B 0,C 180,E1 -18133.635,E2 -18133.635} C_VEL
LIN {X 0,Y 264.291,Z 277.198,A -85,B 0,C 180,E1 -18138.121,E2 -18138.121} C_VEL
LIN {X 0,Y 263.85,Z 274.728,A -85,B 0,C 180,E1 -18142.218,E2 -18142.218} C_VEL
LIN {X 0,Y 263.551,Z 272.869,A -85,B 0,C 180,E1 -18145.943,E2 -18145.943} C_VEL
LIN {X 0,Y 263.311,Z 271.457,A -85,B 0,C 180,E1 -18149.526,E2 -18149.526} C_VEL
LIN {X 0,Y 263.206,Z 270.748,A -85,B 0,C 180,E1 -18151.779,E2 -18151.779} C_VEL
LIN {X 0,Y 263.224,Z 270.697,A -85,B 0,C 180,E1 -18155.198,E2 -18155.198} C_VEL
LIN {X 0,Y 263.261,Z 270.693,A -85,B 0,C 180,E1 -18159.691,E2 -18159.691} C_VEL
LIN {X 0,Y 263.341,Z 270.684,A -85,B 0,C 180,E1 -18164.52,E2 -18164.52} C_VEL
LIN {X 0,Y 263.37,Z 270.68,A -85,B 0,C 180,E1 -18169.232,E2 -18169.232} C_VEL
LIN {X 0,Y 263.568,Z 270.709,A -85,B 0,C 180,E1 -18172.337,E2 -18172.337} C_VEL
LIN {X 0,Y 264.072,Z 272.758,A -85,B 0,C 180,E1 -18178.473,E2 -18178.473} C_VEL
LIN {X 0,Y 264.276,Z 273.386,A -85,B 0,C 180,E1 -18179.998,E2 -18179.998} C_VEL
LIN {X 0,Y 264.229,Z 275.691,A -85,B 0,C 180,E1 -18184.575,E2 -18184.575} C_VEL
LIN {X 0,Y 264.364,Z 277.427,A -85,B 0,C 180,E1 -18187.637,E2 -18187.637} C_VEL
LIN {X 0,Y 264.215,Z 279.4,A -85,B 0,C 180,E1 -18190.729,E2 -18190.729} C_VEL
LIN {X 0,Y 263.745,Z 281.934,A -85,B 0,C 180,E1 -18194.268,E2 -18194.268} C_VEL
LIN {X 0,Y 264.8,Z 285.008,A -85,B 0,C 180,E1 -18194.651,E2 -18194.651} C_VEL
LIN {X 0,Y 265.886,Z 287.034,A -85,B 0,C 180,E1 -18194.982,E2 -18194.982} C_VEL
LIN {X 0,Y 270.705,Z 299.159,A -85,B 0,C 180,E1 -18196.786,E2 -18196.786} C_VEL
LIN {X 0,Y 274.088,Z 311.043,A -85,B 0,C 180,E1 -18198.572,E2 -18198.572} C_VEL
LIN {X 0,Y 275.866,Z 320.854,A -85,B 0,C 180,E1 -18200.114,E2 -18200.114} C_VEL
LIN {X 0,Y 276.578,Z 328.849,A -85,B 0,C 180,E1 -18201.423,E2 -18201.423} C_VEL
LIN {X 0,Y 274.099,Z 339.741,A -85,B 0,C 180,E1 -18203.099,E2 -18203.099} C_VEL
LIN {X 0,Y 271.521,Z 349.845,A -85,B 0,C 180,E1 -18205.054,E2 -18205.054} C_VEL
LIN {X 0,Y 268.958,Z 359.04,A -85,B 0,C 180,E1 -18207.325,E2 -18207.325} C_VEL
LIN {X 0,Y 266.766,Z 366.378,A -85,B 0,C 180,E1 -18209.615,E2 -18209.615} C_VEL
LIN {X 0,Y 264.883,Z 372.52,A -85,B 0,C 180,E1 -18212.047,E2 -18212.047} C_VEL
LIN {X 0,Y 263.587,Z 376.833,A -85,B 0,C 180,E1 -18214.256,E2 -18214.256} C_VEL
LIN {X 0,Y 262.522,Z 380.267,A -85,B 0,C 180,E1 -18216.571,E2 -18216.571} C_VEL
LIN {X 0,Y 261.754,Z 382.668,A -85,B 0,C 180,E1 -18218.865,E2 -18218.865} C_VEL
LIN {X 0,Y 261.184,Z 384.135,A -85,B 0,C 180,E1 -18221.113,E2 -18221.113} C_VEL
LIN {X 0,Y 260.863,Z 384.759,A -85,B 0,C 180,E1 -18223.331,E2 -18223.331} C_VEL
LIN {X 0,Y 260.726,Z 384.593,A -85,B 0,C 180,E1 -18225.507,E2 -18225.507} C_VEL
LIN {X 0,Y 260.721,Z 383.652,A -85,B 0,C 180,E1 -18227.632,E2 -18227.632} C_VEL
LIN {X 0,Y 260.858,Z 381.965,A -85,B 0,C 180,E1 -18229.715,E2 -18229.715} C_VEL
LIN {X 0,Y 261.246,Z 379.549,A -85,B 0,C 180,E1 -18231.777,E2 -18231.777} C_VEL
LIN {X 0,Y 261.676,Z 376.438,A -85,B 0,C 180,E1 -18233.782,E2 -18233.782} C_VEL
LIN {X 0,Y 262.359,Z 371.677,A -85,B 0,C 180,E1 -18236.138,E2 -18236.138} C_VEL
LIN {X 0,Y 263.342,Z 365.131,A -85,B 0,C 180,E1 -18238.646,E2 -18238.646} C_VEL
LIN {X 0,Y 264.552,Z 357.84,A -85,B 0,C 180,E1 -18240.867,E2 -18240.867} C_VEL
LIN {X 0,Y 266.046,Z 348.685,A -85,B 0,C 180,E1 -18243.104,E2 -18243.104} C_VEL
LIN {X 0,Y 267.643,Z 338.085,A -85,B 0,C 180,E1 -18245.157,E2 -18245.157} C_VEL
LIN {X 0,Y 269.25,Z 327.469,A -85,B 0,C 180,E1 -18246.796,E2 -18246.796} C_VEL
LIN {X 0,Y 270.045,Z 319.401,A -85,B 0,C 180,E1 -18247.83,E2 -18247.83} C_VEL
LIN {X 0,Y 268.233,Z 307.417,A -85,B 0,C 180,E1 -18249.286,E2 -18249.286} C_VEL
LIN {X 0,Y 265.704,Z 294.665,A -85,B 0,C 180,E1 -18250.543,E2 -18250.543} C_VEL
LIN {X 0,Y 262.485,Z 281.662,A -85,B 0,C 180,E1 -18251.563,E2 -18251.563} C_VEL
LIN {X 0,Y 262.164,Z 279.938,A -85,B 0,C 180,E1 -18251.691,E2 -18251.691} C_VEL
LIN {X 0,Y 262.627,Z 275.828,A -85,B 0,C 180,E1 -18256.064,E2 -18256.064} C_VEL
LIN {X 0,Y 263.268,Z 271,A -85,B 0,C 180,E1 -18261.403,E2 -18261.403} C_VEL
LIN {X 0,Y 263.407,Z 270.675,A -85,B 0,C 180,E1 -18262.334,E2 -18262.334} C_VEL
LIN {X 0,Y 263.552,Z 270.656,A -85,B 0,C 180,E1 -18266.943,E2 -18266.943} C_VEL
LIN {X 0,Y 263.803,Z 270.623,A -85,B 0,C 180,E1 -18270,E2 -18270} C_VEL
LIN {X 0,Y 263.56,Z 270.654,A -85,B 0,C 180,E1 -18273.057,E2 -18273.057} C_VEL
LIN {X 0,Y 263.563,Z 270.654,A -85,B 0,C 180,E1 -18277.662,E2 -18277.662} C_VEL
LIN {X 0,Y 263.365,Z 270.677,A -85,B 0,C 180,E1 -18280.766,E2 -18280.766} C_VEL
LIN {X 0,Y 263.341,Z 270.68,A -85,B 0,C 180,E1 -18285.478,E2 -18285.478} C_VEL
LIN {X 0,Y 263.26,Z 270.692,A -85,B 0,C 180,E1 -18290.307,E2 -18290.307} C_VEL
LIN {X 0,Y 263.202,Z 270.697,A -85,B 0,C 180,E1 -18295.292,E2 -18295.292} C_VEL
LIN {X 0,Y 263.157,Z 270.698,A -85,B 0,C 180,E1 -18298.732,E2 -18298.732} C_VEL
LIN {X 0,Y 263.125,Z 270.707,A -85,B 0,C 180,E1 -18302.289,E2 -18302.289} C_VEL
LIN {X 0,Y 263.181,Z 270.701,A -85,B 0,C 180,E1 -18305.978,E2 -18305.978} C_VEL
LIN {X 0,Y 263.153,Z 270.699,A -85,B 0,C 180,E1 -18309.863,E2 -18309.863} C_VEL
LIN {X 0,Y 263.183,Z 270.696,A -85,B 0,C 180,E1 -18313.866,E2 -18313.866} C_VEL
LIN {X 0,Y 263.204,Z 270.696,A -85,B 0,C 180,E1 -18318.386,E2 -18318.386} C_VEL
LIN {X 0,Y 263.196,Z 270.7,A -85,B 0,C 180,E1 -18323.232,E2 -18323.232} C_VEL
LIN {X 0,Y 263.176,Z 270.695,A -85,B 0,C 180,E1 -18325.892,E2 -18325.892} C_VEL
LIN {X 0,Y 263.143,Z 270.695,A -85,B 0,C 180,E1 -18329.508,E2 -18329.508} C_VEL
LIN {X 0,Y 263.186,Z 270.698,A -85,B 0,C 180,E1 -18333.004,E2 -18333.004} C_VEL
LIN {X 0,Y 263.177,Z 270.701,A -85,B 0,C 180,E1 -18336.389,E2 -18336.389} C_VEL
LIN {X 0,Y 263.257,Z 270.69,A -85,B 0,C 180,E1 -18339.695,E2 -18339.695} C_VEL
LIN {X 0,Y 263.339,Z 270.679,A -85,B 0,C 180,E1 -18344.523,E2 -18344.523} C_VEL
LIN {X 0,Y 263.35,Z 270.671,A -85,B 0,C 180,E1 -18349.235,E2 -18349.235} C_VEL
LIN {X 0,Y 263.553,Z 270.653,A -85,B 0,C 180,E1 -18352.34,E2 -18352.34} C_VEL
LIN {X 0,Y 263.747,Z 270.631,A -85,B 0,C 180,E1 -18358.475,E2 -18358.475} C_VEL
LIN {X 0,Y 263.748,Z 270.627,A -85,B 0,C 180,E1 -18361.529,E2 -18361.529} C_VEL
LIN {X 0,Y 263.57,Z 270.648,A -85,B 0,C 180,E1 -18367.663,E2 -18367.663} C_VEL
LIN {X 0,Y 263.372,Z 270.676,A -85,B 0,C 180,E1 -18370.767,E2 -18370.767} C_VEL
LIN {X 0,Y 263.344,Z 270.68,A -85,B 0,C 180,E1 -18375.48,E2 -18375.48} C_VEL
LIN {X 0,Y 263.263,Z 270.688,A -85,B 0,C 180,E1 -18380.308,E2 -18380.308} C_VEL
LIN {X 0,Y 263.197,Z 270.698,A -85,B 0,C 180,E1 -18384.359,E2 -18384.359} C_VEL
LIN {X 0,Y 262.559,Z 270.78,A -85,B 0,C 180,E1 -18385.637,E2 -18385.637} C_VEL
LIN {X 0,Y 259.655,Z 271.139,A -85,B 0,C 180,E1 -18387.718,E2 -18387.718} C_VEL
LIN {X 0,Y 257.181,Z 271.449,A -85,B 0,C 180,E1 -18389.411,E2 -18389.411} C_VEL
LIN {X 0,Y 256.147,Z 271.577,A -85,B 0,C 180,E1 -18390.726,E2 -18390.726} C_VEL
LIN {X 0,Y 256.08,Z 271.587,A -85,B 0,C 180,E1 -18391.171,E2 -18391.171} C_VEL
LIN {X 0,Y 256.084,Z 271.587,A -85,B 0,C 180,E1 -18395.194,E2 -18395.194} C_VEL
LIN {X 0,Y 256.117,Z 271.584,A -85,B 0,C 180,E1 -18397.272,E2 -18397.272} C_VEL
LIN {X 0,Y 256.057,Z 271.591,A -85,B 0,C 180,E1 -18401.205,E2 -18401.205} C_VEL
LIN {X 0,Y 256.134,Z 271.724,A -85,B 0,C 180,E1 -18404.63,E2 -18404.63} C_VEL
LIN {X 0,Y 256.936,Z 276.141,A -85,B 0,C 180,E1 -18408.969,E2 -18408.969} C_VEL
LIN {X 0,Y 257.468,Z 279.749,A -85,B 0,C 180,E1 -18412.338,E2 -18412.338} C_VEL
LIN {X 0,Y 257.4,Z 282.782,A -85,B 0,C 180,E1 -18415.014,E2 -18415.014} C_VEL
LIN {X 0,Y 256.331,Z 288.121,A -85,B 0,C 180,E1 -18419.521,E2 -18419.521} C_VEL
LIN {X 0,Y 255.614,Z 293.305,A -85,B 0,C 180,E1 -18423.792,E2 -18423.792} C_VEL
LIN {X 0,Y 258.319,Z 307.662,A -85,B 0,C 180,E1 -18424.839,E2 -18424.839} C_VEL
LIN {X 0,Y 260.256,Z 321.098,A -85,B 0,C 180,E1 -18426.105,E2 -18426.105} C_VEL
LIN {X 0,Y 261.478,Z 332.629,A -85,B 0,C 180,E1 -18427.457,E2 -18427.457} C_VEL
LIN {X 0,Y 261.956,Z 340.565,A -85,B 0,C 180,E1 -18428.559,E2 -18428.559} C_VEL
LIN {X 0,Y 260.201,Z 351.721,A -85,B 0,C 180,E1 -18430.268,E2 -18430.268} C_VEL
LIN {X 0,Y 258.568,Z 361.764,A -85,B 0,C 180,E1 -18432.218,E2 -18432.218} C_VEL
LIN {X 0,Y 257.309,Z 369.849,A -85,B 0,C 180,E1 -18434.149,E2 -18434.149} C_VEL
LIN {X 0,Y 255.967,Z 377.876,A -85,B 0,C 180,E1 -18436.504,E2 -18436.504} C_VEL
LIN {X 0,Y 255.049,Z 384.297,A -85,B 0,C 180,E1 -18438.879,E2 -18438.879} C_VEL
LIN {X 0,Y 254.463,Z 389.379,A -85,B 0,C 180,E1 -18441.263,E2 -18441.263} C_VEL
LIN {X 0,Y 254.108,Z 393.294,A -85,B 0,C 180,E1 -18443.648,E2 -18443.648} C_VEL
LIN {X 0,Y 253.979,Z 395.296,A -85,B 0,C 180,E1 -18445.238,E2 -18445.238} C_VEL
LIN {X 0,Y 254.015,Z 396.878,A -85,B 0,C 180,E1 -18446.828,E2 -18446.828} C_VEL
LIN {X 0,Y 254.05,Z 398.034,A -85,B 0,C 180,E1 -18448.415,E2 -18448.415} C_VEL
LIN {X 0,Y 254.057,Z 398.736,A -85,B 0,C 180,E1 -18450,E2 -18450} C_VEL
LIN {X 0,Y 254.017,Z 399.04,A -85,B 0,C 180,E1 -18451.585,E2 -18451.585} C_VEL
LIN {X 0,Y 253.953,Z 398.953,A -85,B 0,C 180,E1 -18453.173,E2 -18453.173} C_VEL
LIN {X 0,Y 253.995,Z 398.335,A -85,B 0,C 180,E1 -18455.038,E2 -18455.038} C_VEL
LIN {X 0,Y 254.338,Z 396.26,A -85,B 0,C 180,E1 -18457.941,E2 -18457.941} C_VEL
LIN {X 0,Y 254.965,Z 393.531,A -85,B 0,C 180,E1 -18460.321,E2 -18460.321} C_VEL
LIN {X 0,Y 255.947,Z 389.808,A -85,B 0,C 180,E1 -18462.689,E2 -18462.689} C_VEL
LIN {X 0,Y 257.338,Z 385.023,A -85,B 0,C 180,E1 -18465.037,E2 -18465.037} C_VEL
LIN {X 0,Y 259.672,Z 377.909,A -85,B 0,C 180,E1 -18467.726,E2 -18467.726} C_VEL
LIN {X 0,Y 261.77,Z 369.931,A -85,B 0,C 180,E1 -18470.113,E2 -18470.113} C_VEL
LIN {X 0,Y 264.416,Z 360.772,A -85,B 0,C 180,E1 -18472.256,E2 -18472.256} C_VEL
LIN {X 0,Y 267.095,Z 351.07,A -85,B 0,C 180,E1 -18474.069,E2 -18474.069} C_VEL
LIN {X 0,Y 268.056,Z 346.601,A -85,B 0,C 180,E1 -18474.802,E2 -18474.802} C_VEL
LIN {X 0,Y 268.074,Z 335.355,A -85,B 0,C 180,E1 -18476.687,E2 -18476.687} C_VEL
LIN {X 0,Y 267.064,Z 324.973,A -85,B 0,C 180,E1 -18478.273,E2 -18478.273} C_VEL
LIN {X 0,Y 264.613,Z 312.934,A -85,B 0,C 180,E1 -18480.019,E2 -18480.019} C_VEL
LIN {X 0,Y 261.52,Z 302.476,A -85,B 0,C 180,E1 -18481.509,E2 -18481.509} C_VEL
LIN {X 0,Y 258.691,Z 295.096,A -85,B 0,C 180,E1 -18482.573,E2 -18482.573} C_VEL
LIN {X 0,Y 257.567,Z 291.813,A -85,B 0,C 180,E1 -18482.994,E2 -18482.994} C_VEL
LIN {X 0,Y 257.531,Z 291.359,A -85,B 0,C 180,E1 -18483.078,E2 -18483.078} C_VEL
LIN {X 0,Y 258.012,Z 289.208,A -85,B 0,C 180,E1 -18485.195,E2 -18485.195} C_VEL
LIN {X 0,Y 258.263,Z 286.62,A -85,B 0,C 180,E1 -18487.89,E2 -18487.89} C_VEL
LIN {X 0,Y 258.086,Z 284.091,A -85,B 0,C 180,E1 -18490.808,E2 -18490.808} C_VEL
LIN {X 0,Y 257.681,Z 280.973,A -85,B 0,C 180,E1 -18494.834,E2 -18494.834} C_VEL
LIN {X 0,Y 257.222,Z 278.167,A -85,B 0,C 180,E1 -18499.022,E2 -18499.022} C_VEL
LIN {X 0,Y 256.9,Z 275.911,A -85,B 0,C 180,E1 -18502.995,E2 -18502.995} C_VEL
LIN {X 0,Y 256.547,Z 274.186,A -85,B 0,C 180,E1 -18506.776,E2 -18506.776} C_VEL
LIN {X 0,Y 256.346,Z 272.859,A -85,B 0,C 180,E1 -18510.428,E2 -18510.428} C_VEL
LIN {X 0,Y 256.187,Z 271.732,A -85,B 0,C 180,E1 -18514.86,E2 -18514.86} C_VEL
LIN {X 0,Y 256.164,Z 271.577,A -85,B 0,C 180,E1 -18519.103,E2 -18519.103} C_VEL
LIN {X 0,Y 256.291,Z 271.561,A -85,B 0,C 180,E1 -18524.083,E2 -18524.083} C_VEL
LIN {X 0,Y 256.332,Z 271.636,A -85,B 0,C 180,E1 -18528.933,E2 -18528.933} C_VEL
LIN {X 0,Y 256.631,Z 272.271,A -85,B 0,C 180,E1 -18532.128,E2 -18532.128} C_VEL
LIN {X 0,Y 256.9,Z 273.713,A -85,B 0,C 180,E1 -18536.862,E2 -18536.862} C_VEL
LIN {X 0,Y 257.349,Z 274.876,A -85,B 0,C 180,E1 -18539.998,E2 -18539.998} C_VEL
LIN {X 0,Y 257.296,Z 276.362,A -85,B 0,C 180,E1 -18543.13,E2 -18543.13} C_VEL
LIN {X 0,Y 257.355,Z 278.401,A -85,B 0,C 180,E1 -18546.955,E2 -18546.955} C_VEL
LIN {X 0,Y 257.276,Z 280.507,A -85,B 0,C 180,E1 -18550.458,E2 -18550.458} C_VEL
LIN {X 0,Y 256.909,Z 282.339,A -85,B 0,C 180,E1 -18552.941,E2 -18552.941} C_VEL
LIN {X 0,Y 258.056,Z 285.445,A -85,B 0,C 180,E1 -18553.383,E2 -18553.383} C_VEL
LIN {X 0,Y 259.221,Z 287.69,A -85,B 0,C 180,E1 -18553.771,E2 -18553.771} C_VEL
LIN {X 0,Y 262.352,Z 294.891,A -85,B 0,C 180,E1 -18554.939,E2 -18554.939} C_VEL
LIN {X 0,Y 266.09,Z 305.742,A -85,B 0,C 180,E1 -18556.69,E2 -18556.69} C_VEL
LIN {X 0,Y 268.744,Z 316.783,A -85,B 0,C 180,E1 -18558.485,E2 -18558.485} C_VEL
LIN {X 0,Y 270.085,Z 326.678,A -85,B 0,C 180,E1 -18560.173,E2 -18560.173} C_VEL
LIN {X 0,Y 270.287,Z 329.681,A -85,B 0,C 180,E1 -18560.705,E2 -18560.705} C_VEL
LIN {X 0,Y 267.602,Z 341.203,A -85,B 0,C 180,E1 -18562.566,E2 -18562.566} C_VEL
LIN {X 0,Y 265.035,Z 350.681,A -85,B 0,C 180,E1 -18564.475,E2 -18564.475} C_VEL
LIN {X 0,Y 262.495,Z 359.221,A -85,B 0,C 180,E1 -18566.642,E2 -18566.642} C_VEL
LIN {X 0,Y 260.077,Z 366.904,A -85,B 0,C 180,E1 -18569.102,E2 -18569.102} C_VEL
LIN {X 0,Y 258.028,Z 373.123,A -85,B 0,C 180,E1 -18571.677,E2 -18571.677} C_VEL
LIN {X 0,Y 256.292,Z 378.429,A -85,B 0,C 180,E1 -18574.651,E2 -18574.651} C_VEL
LIN {X 0,Y 255.158,Z 381.769,A -85,B 0,C 180,E1 -18577.295,E2 -18577.295} C_VEL
LIN {X 0,Y 254.489,Z 383.568,A -85,B 0,C 180,E1 -18579.43,E2 -18579.43} C_VEL
LIN {X 0,Y 253.993,Z 384.68,A -85,B 0,C 180,E1 -18581.662,E2 -18581.662} C_VEL
LIN {X 0,Y 253.725,Z 385.014,A -85,B 0,C 180,E1 -18583.932,E2 -18583.932} C_VEL
LIN {X 0,Y 253.613,Z 384.527,A -85,B 0,C 180,E1 -18586.15,E2 -18586.15} C_VEL
LIN {X 0,Y 253.644,Z 383.219,A -85,B 0,C 180,E1 -18588.424,E2 -18588.424} C_VEL
LIN {X 0,Y 253.936,Z 380.959,A -85,B 0,C 180,E1 -18590.795,E2 -18590.795} C_VEL
LIN {X 0,Y 254.429,Z 377.622,A -85,B 0,C 180,E1 -18593.227,E2 -18593.227} C_VEL
LIN {X 0,Y 255.118,Z 372.999,A -85,B 0,C 180,E1 -18595.731,E2 -18595.731} C_VEL
LIN {X 0,Y 256.063,Z 366.857,A -85,B 0,C 180,E1 -18598.299,E2 -18598.299} C_VEL
LIN {X 0,Y 257.203,Z 360.069,A -85,B 0,C 180,E1 -18600.539,E2 -18600.539} C_VEL
LIN {X 0,Y 258.574,Z 351.777,A -85,B 0,C 180,E1 -18602.744,E2 -18602.744} C_VEL
LIN {X 0,Y 260.096,Z 342.154,A -85,B 0,C 180,E1 -18604.814,E2 -18604.814} C_VEL
LIN {X 0,Y 261.636,Z 332.739,A -85,B 0,C 180,E1 -18606.45,E2 -18606.45} C_VEL
LIN {X 0,Y 263.202,Z 321.275,A -85,B 0,C 180,E1 -18608.049,E2 -18608.049} C_VEL
LIN {X 0,Y 261.821,Z 310.987,A -85,B 0,C 180,E1 -18609.372,E2 -18609.372} C_VEL
LIN {X 0,Y 259.67,Z 299.297,A -85,B 0,C 180,E1 -18610.638,E2 -18610.638} C_VEL
LIN {X 0,Y 256.613,Z 286.177,A -85,B 0,C 180,E1 -18611.797,E2 -18611.797} C_VEL
LIN {X 0,Y 255.152,Z 280.135,A -85,B 0,C 180,E1 -18612.26,E2 -18612.26} C_VEL
LIN {X 0,Y 255.512,Z 276.994,A -85,B 0,C 180,E1 -18615.668,E2 -18615.668} C_VEL
LIN {X 0,Y 256.173,Z 272.28,A -85,B 0,C 180,E1 -18620.968,E2 -18620.968} C_VEL
LIN {X 0,Y 256.349,Z 271.554,A -85,B 0,C 180,E1 -18622.122,E2 -18622.122} C_VEL
LIN {X 0,Y 256.312,Z 271.557,A -85,B 0,C 180,E1 -18625.282,E2 -18625.282} C_VEL
LIN {X 0,Y 256.705,Z 271.509,A -85,B 0,C 180,E1 -18628.431,E2 -18628.431} C_VEL
LIN {X 0,Y 256.708,Z 271.506,A -85,B 0,C 180,E1 -18631.569,E2 -18631.569} C_VEL
LIN {X 0,Y 256.53,Z 271.531,A -85,B 0,C 180,E1 -18637.873,E2 -18637.873} C_VEL
LIN {X 0,Y 256.301,Z 271.556,A -85,B 0,C 180,E1 -18641.066,E2 -18641.066} C_VEL
LIN {X 0,Y 256.291,Z 271.561,A -85,B 0,C 180,E1 -18645.915,E2 -18645.915} C_VEL
LIN {X 0,Y 256.21,Z 271.568,A -85,B 0,C 180,E1 -18650.891,E2 -18650.891} C_VEL
LIN {X 0,Y 256.182,Z 271.571,A -85,B 0,C 180,E1 -18655.14,E2 -18655.14} C_VEL
LIN {X 0,Y 256.095,Z 271.58,A -85,B 0,C 180,E1 -18659.602,E2 -18659.602} C_VEL
LIN {X 0,Y 256.076,Z 271.586,A -85,B 0,C 180,E1 -18663.291,E2 -18663.291} C_VEL
LIN {X 0,Y 256.133,Z 271.579,A -85,B 0,C 180,E1 -18667.28,E2 -18667.28} C_VEL
LIN {X 0,Y 256.124,Z 271.574,A -85,B 0,C 180,E1 -18671.189,E2 -18671.189} C_VEL
LIN {X 0,Y 256.108,Z 271.581,A -85,B 0,C 180,E1 -18675.518,E2 -18675.518} C_VEL
LIN {X 0,Y 256.124,Z 271.58,A -85,B 0,C 180,E1 -18678.813,E2 -18678.813} C_VEL
LIN {X 0,Y 256.146,Z 271.577,A -85,B 0,C 180,E1 -18682.873,E2 -18682.873} C_VEL
LIN {X 0,Y 256.078,Z 271.58,A -85,B 0,C 180,E1 -18686.711,E2 -18686.711} C_VEL
LIN {X 0,Y 256.131,Z 271.573,A -85,B 0,C 180,E1 -18691.406,E2 -18691.406} C_VEL
LIN {X 0,Y 256.161,Z 271.573,A -85,B 0,C 180,E1 -18695.701,E2 -18695.701} C_VEL
LIN {X 0,Y 256.161,Z 271.576,A -85,B 0,C 180,E1 -18699.107,E2 -18699.107} C_VEL
LIN {X 0,Y 256.289,Z 271.555,A -85,B 0,C 180,E1 -18704.086,E2 -18704.086} C_VEL
LIN {X 0,Y 256.288,Z 271.546,A -85,B 0,C 180,E1 -18707.33,E2 -18707.33} C_VEL
LIN {X 0,Y 256.51,Z 271.528,A -85,B 0,C 180,E1 -18712.128,E2 -18712.128} C_VEL
LIN {X 0,Y 256.495,Z 271.534,A -85,B 0,C 180,E1 -18716.86,E2 -18716.86} C_VEL
LIN {X 0,Y 256.762,Z 271.501,A -85,B 0,C 180,E1 -18720.002,E2 -18720.002} C_VEL
LIN {X 0,Y 256.496,Z 271.526,A -85,B 0,C 180,E1 -18723.143,E2 -18723.143} C_VEL
LIN {X 0,Y 256.538,Z 271.525,A -85,B 0,C 180,E1 -18727.875,E2 -18727.875} C_VEL
LIN {X 0,Y 256.308,Z 271.556,A -85,B 0,C 180,E1 -18731.068,E2 -18731.068} C_VEL
LIN {X 0,Y 256.279,Z 271.56,A -85,B 0,C 180,E1 -18735.918,E2 -18735.918} C_VEL
LIN {X 0,Y 256.166,Z 271.572,A -85,B 0,C 180,E1 -18740.897,E2 -18740.897} C_VEL
LIN {X 0,Y 256.188,Z 271.572,A -85,B 0,C 180,E1 -18745.14,E2 -18745.14} C_VEL
LIN {X 0,Y 256.111,Z 271.584,A -85,B 0,C 180,E1 -18749.602,E2 -18749.602} C_VEL
LIN {X 0,Y 256.08,Z 271.587,A -85,B 0,C 180,E1 -18751.171,E2 -18751.171} C_VEL
LIN {X 0,Y 255.459,Z 271.672,A -85,B 0,C 180,E1 -18752.484,E2 -18752.484} C_VEL
LIN {X 0,Y 252.627,Z 272.025,A -85,B 0,C 180,E1 -18754.624,E2 -18754.624} C_VEL
LIN {X 0,Y 250.186,Z 272.324,A -85,B 0,C 180,E1 -18756.365,E2 -18756.365} C_VEL
LIN {X 0,Y 249.124,Z 272.454,A -85,B 0,C 180,E1 -18757.716,E2 -18757.716} C_VEL
LIN {X 0,Y 249.032,Z 272.464,A -85,B 0,C 180,E1 -18758.174,E2 -18758.174} C_VEL
LIN {X 0,Y 249.013,Z 272.468,A -85,B 0,C 180,E1 -18762.794,E2 -18762.794} C_VEL
LIN {X 0,Y 249.044,Z 272.516,A -85,B 0,C 180,E1 -18764.31,E2 -18764.31} C_VEL
LIN {X 0,Y 249.624,Z 275.626,A -85,B 0,C 180,E1 -18767.492,E2 -18767.492} C_VEL
LIN {X 0,Y 250.253,Z 279.011,A -85,B 0,C 180,E1 -18770.813,E2 -18770.813} C_VEL
LIN {X 0,Y 250.457,Z 282.331,A -85,B 0,C 180,E1 -18773.895,E2 -18773.895} C_VEL
LIN {X 0,Y 249.902,Z 285.564,A -85,B 0,C 180,E1 -18776.744,E2 -18776.744} C_VEL
LIN {X 0,Y 248.905,Z 290.887,A -85,B 0,C 180,E1 -18781.315,E2 -18781.315} C_VEL
LIN {X 0,Y 248.603,Z 293.109,A -85,B 0,C 180,E1 -18783.197,E2 -18783.197} C_VEL
LIN {X 0,Y 251.425,Z 308.085,A -85,B 0,C 180,E1 -18784.346,E2 -18784.346} C_VEL
LIN {X 0,Y 253.375,Z 321.549,A -85,B 0,C 180,E1 -18785.674,E2 -18785.674} C_VEL
LIN {X 0,Y 254.461,Z 332.588,A -85,B 0,C 180,E1 -18787.016,E2 -18787.016} C_VEL
LIN {X 0,Y 255.004,Z 340.548,A -85,B 0,C 180,E1 -18788.157,E2 -18788.157} C_VEL
LIN {X 0,Y 253.517,Z 350.551,A -85,B 0,C 180,E1 -18789.725,E2 -18789.725} C_VEL
LIN {X 0,Y 252.009,Z 359.685,A -85,B 0,C 180,E1 -18791.48,E2 -18791.48} C_VEL
LIN {X 0,Y 250.448,Z 369.001,A -85,B 0,C 180,E1 -18793.703,E2 -18793.703} C_VEL
LIN {X 0,Y 249.045,Z 377.134,A -85,B 0,C 180,E1 -18796.121,E2 -18796.121} C_VEL
LIN {X 0,Y 248.059,Z 383.678,A -85,B 0,C 180,E1 -18798.561,E2 -18798.561} C_VEL
LIN {X 0,Y 247.406,Z 388.858,A -85,B 0,C 180,E1 -18801.011,E2 -18801.011} C_VEL
LIN {X 0,Y 247.037,Z 392.856,A -85,B 0,C 180,E1 -18803.466,E2 -18803.466} C_VEL
LIN {X 0,Y 246.888,Z 394.897,A -85,B 0,C 180,E1 -18805.101,E2 -18805.101} C_VEL
LIN {X 0,Y 246.912,Z 396.516,A -85,B 0,C 180,E1 -18806.736,E2 -18806.736} C_VEL
LIN {X 0,Y 246.958,Z 397.721,A -85,B 0,C 180,E1 -18808.369,E2 -18808.369} C_VEL
LIN {X 0,Y 246.986,Z 398.481,A -85,B 0,C 180,E1 -18810,E2 -18810} C_VEL
LIN {X 0,Y 246.924,Z 398.819,A -85,B 0,C 180,E1 -18811.631,E2 -18811.631} C_VEL
LIN {X 0,Y 246.888,Z 398.328,A -85,B 0,C 180,E1 -18814.899,E2 -18814.899} C_VEL
LIN {X 0,Y 247.018,Z 397.48,A -85,B 0,C 180,E1 -18816.534,E2 -18816.534} C_VEL
LIN {X 0,Y 247.702,Z 394.548,A -85,B 0,C 180,E1 -18819.801,E2 -18819.801} C_VEL
LIN {X 0,Y 248.624,Z 391.252,A -85,B 0,C 180,E1 -18822.24,E2 -18822.24} C_VEL
LIN {X 0,Y 249.886,Z 386.925,A -85,B 0,C 180,E1 -18824.662,E2 -18824.662} C_VEL
LIN {X 0,Y 252.174,Z 380.436,A -85,B 0,C 180,E1 -18827.433,E2 -18827.433} C_VEL
LIN {X 0,Y 254.054,Z 373.871,A -85,B 0,C 180,E1 -18829.661,E2 -18829.661} C_VEL
LIN {X 0,Y 256.864,Z 364.743,A -85,B 0,C 180,E1 -18832.098,E2 -18832.098} C_VEL
LIN {X 0,Y 259.529,Z 355.972,A -85,B 0,C 180,E1 -18833.965,E2 -18833.965} C_VEL
LIN {X 0,Y 261.546,Z 348.722,A -85,B 0,C 180,E1 -18835.25,E2 -18835.25} C_VEL
LIN {X 0,Y 261.83,Z 338.057,A -85,B 0,C 180,E1 -18837.149,E2 -18837.149} C_VEL
LIN {X 0,Y 261.157,Z 328.42,A -85,B 0,C 180,E1 -18838.72,E2 -18838.72} C_VEL
LIN {X 0,Y 259.056,Z 316.462,A -85,B 0,C 180,E1 -18840.606,E2 -18840.606} C_VEL
LIN {X 0,Y 256.754,Z 307.638,A -85,B 0,C 180,E1 -18841.943,E2 -18841.943} C_VEL
LIN {X 0,Y 253.518,Z 298.564,A -85,B 0,C 180,E1 -18843.378,E2 -18843.378} C_VEL
LIN {X 0,Y 252.109,Z 295.031,A -85,B 0,C 180,E1 -18843.929,E2 -18843.929} C_VEL
LIN {X 0,Y 250.931,Z 291.938,A -85,B 0,C 180,E1 -18844.393,E2 -18844.393} C_VEL
LIN {X 0,Y 250.805,Z 291.126,A -85,B 0,C 180,E1 -18844.49,E2 -18844.49} C_VEL
LIN {X 0,Y 251.29,Z 287.844,A -85,B 0,C 180,E1 -18847.972,E2 -18847.972} C_VEL
LIN {X 0,Y 251.123,Z 285.375,A -85,B 0,C 180,E1 -18850.917,E2 -18850.917} C_VEL
LIN {X 0,Y 250.757,Z 282.689,A -85,B 0,C 180,E1 -18854.48,E2 -18854.48} C_VEL
LIN {X 0,Y 250.443,Z 280.55,A -85,B 0,C 180,E1 -18857.661,E2 -18857.661} C_VEL
LIN {X 0,Y 250.064,Z 278.088,A -85,B 0,C 180,E1 -18861.898,E2 -18861.898} C_VEL
LIN {X 0,Y 249.715,Z 276.263,A -85,B 0,C 180,E1 -18865.743,E2 -18865.743} C_VEL
LIN {X 0,Y 249.446,Z 274.419,A -85,B 0,C 180,E1 -18870.854,E2 -18870.854} C_VEL
LIN {X 0,Y 249.298,Z 273.42,A -85,B 0,C 180,E1 -18874.982,E2 -18874.982} C_VEL
LIN {X 0,Y 249.16,Z 272.939,A -85,B 0,C 180,E1 -18878.56,E2 -18878.56} C_VEL
LIN {X 0,Y 249.27,Z 272.767,A -85,B 0,C 180,E1 -18883.622,E2 -18883.622} C_VEL
LIN {X 0,Y 249.418,Z 273.239,A -85,B 0,C 180,E1 -18888.622,E2 -18888.622} C_VEL
LIN {X 0,Y 249.694,Z 273.846,A -85,B 0,C 180,E1 -18891.908,E2 -18891.908} C_VEL
LIN {X 0,Y 249.967,Z 275.232,A -85,B 0,C 180,E1 -18896.775,E2 -18896.775} C_VEL
LIN {X 0,Y 250.428,Z 276.382,A -85,B 0,C 180,E1 -18899.998,E2 -18899.998} C_VEL
LIN {X 0,Y 250.342,Z 278.661,A -85,B 0,C 180,E1 -18904.829,E2 -18904.829} C_VEL
LIN {X 0,Y 250.4,Z 280.398,A -85,B 0,C 180,E1 -18908.065,E2 -18908.065} C_VEL
LIN {X 0,Y 250.25,Z 281.924,A -85,B 0,C 180,E1 -18910.607,E2 -18910.607} C_VEL
LIN {X 0,Y 250.115,Z 282.456,A -85,B 0,C 180,E1 -18911.444,E2 -18911.444} C_VEL
LIN {X 0,Y 251.19,Z 285.623,A -85,B 0,C 180,E1 -18911.926,E2 -18911.926} C_VEL
LIN {X 0,Y 252.476,Z 287.774,A -85,B 0,C 180,E1 -18912.367,E2 -18912.367} C_VEL
LIN {X 0,Y 256.999,Z 298.34,A -85,B 0,C 180,E1 -18914.246,E2 -18914.246} C_VEL
LIN {X 0,Y 260.428,Z 308.867,A -85,B 0,C 180,E1 -18916.056,E2 -18916.056} C_VEL
LIN {X 0,Y 262.74,Z 319.519,A -85,B 0,C 180,E1 -18917.913,E2 -18917.913} C_VEL
LIN {X 0,Y 263.911,Z 329.602,A -85,B 0,C 180,E1 -18919.745,E2 -18919.745} C_VEL
LIN {X 0,Y 263.592,Z 333.517,A -85,B 0,C 180,E1 -18920.421,E2 -18920.421} C_VEL
LIN {X 0,Y 260.924,Z 343.503,A -85,B 0,C 180,E1 -18922.151,E2 -18922.151} C_VEL
LIN {X 0,Y 258.278,Z 352.462,A -85,B 0,C 180,E1 -18924.087,E2 -18924.087} C_VEL
LIN {X 0,Y 255.446,Z 361.322,A -85,B 0,C 180,E1 -18926.487,E2 -18926.487} C_VEL
LIN {X 0,Y 252.905,Z 368.789,A -85,B 0,C 180,E1 -18929.096,E2 -18929.096} C_VEL
LIN {X 0,Y 250.875,Z 374.517,A -85,B 0,C 180,E1 -18931.683,E2 -18931.683} C_VEL
LIN {X 0,Y 249.35,Z 378.907,A -85,B 0,C 180,E1 -18934.31,E2 -18934.31} C_VEL
LIN {X 0,Y 247.997,Z 382.57,A -85,B 0,C 180,E1 -18937.489,E2 -18937.489} C_VEL
LIN {X 0,Y 247.058,Z 384.731,A -85,B 0,C 180,E1 -18940.862,E2 -18940.862} C_VEL
LIN {X 0,Y 246.695,Z 385.199,A -85,B 0,C 180,E1 -18943.132,E2 -18943.132} C_VEL
LIN {X 0,Y 246.524,Z 384.903,A -85,B 0,C 180,E1 -18945.453,E2 -18945.453} C_VEL
LIN {X 0,Y 246.516,Z 383.771,A -85,B 0,C 180,E1 -18947.834,E2 -18947.834} C_VEL
LIN {X 0,Y 246.742,Z 381.716,A -85,B 0,C 180,E1 -18950.265,E2 -18950.265} C_VEL
LIN {X 0,Y 247.369,Z 377.645,A -85,B 0,C 180,E1 -18953.372,E2 -18953.372} C_VEL
LIN {X 0,Y 248.087,Z 372.899,A -85,B 0,C 180,E1 -18955.98,E2 -18955.98} C_VEL
LIN {X 0,Y 249.163,Z 366.323,A -85,B 0,C 180,E1 -18958.739,E2 -18958.739} C_VEL
LIN {X 0,Y 250.364,Z 359.284,A -85,B 0,C 180,E1 -18961.061,E2 -18961.061} C_VEL
LIN {X 0,Y 251.943,Z 350.097,A -85,B 0,C 180,E1 -18963.493,E2 -18963.493} C_VEL
LIN {X 0,Y 253.436,Z 341.027,A -85,B 0,C 180,E1 -18965.421,E2 -18965.421} C_VEL
LIN {X 0,Y 255.302,Z 329.717,A -85,B 0,C 180,E1 -18967.333,E2 -18967.333} C_VEL
LIN {X 0,Y 256.27,Z 321.512,A -85,B 0,C 180,E1 -18968.482,E2 -18968.482} C_VEL
LIN {X 0,Y 254.606,Z 309.798,A -85,B 0,C 180,E1 -18970.026,E2 -18970.026} C_VEL
LIN {X 0,Y 252.246,Z 297.545,A -85,B 0,C 180,E1 -18971.371,E2 -18971.371} C_VEL
LIN {X 0,Y 249.154,Z 284.607,A -85,B 0,C 180,E1 -18972.508,E2 -18972.508} C_VEL
LIN {X 0,Y 248.145,Z 280.304,A -85,B 0,C 180,E1 -18972.859,E2 -18972.859} C_VEL
LIN {X 0,Y 248.55,Z 276.687,A -85,B 0,C 180,E1 -18976.927,E2 -18976.927} C_VEL
LIN {X 0,Y 249.253,Z 272.438,A -85,B 0,C 180,E1 -18981.896,E2 -18981.896} C_VEL
LIN {X 0,Y 249.377,Z 272.418,A -85,B 0,C 180,E1 -18983.528,E2 -18983.528} C_VEL
LIN {X 0,Y 249.666,Z 272.386,A -85,B 0,C 180,E1 -18988.387,E2 -18988.387} C_VEL
LIN {X 0,Y 249.67,Z 272.383,A -85,B 0,C 180,E1 -18991.613,E2 -18991.613} C_VEL
LIN {X 0,Y 249.452,Z 272.415,A -85,B 0,C 180,E1 -18996.471,E2 -18996.471} C_VEL
LIN {X 0,Y 249.415,Z 272.416,A -85,B 0,C 180,E1 -18999.734,E2 -18999.734} C_VEL
LIN {X 0,Y 249.197,Z 272.443,A -85,B 0,C 180,E1 -19004.704,E2 -19004.704} C_VEL
LIN {X 0,Y 249.131,Z 272.449,A -85,B 0,C 180,E1 -19008.078,E2 -19008.078} C_VEL
LIN {X 0,Y 249.097,Z 272.455,A -85,B 0,C 180,E1 -19011.517,E2 -19011.517} C_VEL
LIN {X 0,Y 249.124,Z 272.451,A -85,B 0,C 180,E1 -19015.484,E2 -19015.484} C_VEL
LIN {X 0,Y 249.064,Z 272.452,A -85,B 0,C 180,E1 -19018.99,E2 -19018.99} C_VEL
LIN {X 0,Y 249.027,Z 272.463,A -85,B 0,C 180,E1 -19022.426,E2 -19022.426} C_VEL
LIN {X 0,Y 249.067,Z 272.457,A -85,B 0,C 180,E1 -19026.339,E2 -19026.339} C_VEL
LIN {X 0,Y 249.075,Z 272.449,A -85,B 0,C 180,E1 -19030.464,E2 -19030.464} C_VEL
LIN {X 0,Y 249.085,Z 272.445,A -85,B 0,C 180,E1 -19032.815,E2 -19032.815} C_VEL
LIN {X 0,Y 249.09,Z 272.457,A -85,B 0,C 180,E1 -19037.382,E2 -19037.382} C_VEL
LIN {X 0,Y 249.045,Z 272.462,A -85,B 0,C 180,E1 -19041.626,E2 -19041.626} C_VEL
LIN {X 0,Y 249.054,Z 272.454,A -85,B 0,C 180,E1 -19045.644,E2 -19045.644} C_VEL
LIN {X 0,Y 249.045,Z 272.449,A -85,B 0,C 180,E1 -19049.475,E2 -19049.475} C_VEL
LIN {X 0,Y 249.067,Z 272.457,A -85,B 0,C 180,E1 -19053.164,E2 -19053.164} C_VEL
LIN {X 0,Y 249.073,Z 272.46,A -85,B 0,C 180,E1 -19056.734,E2 -19056.734} C_VEL
LIN {X 0,Y 249.105,Z 272.454,A -85,B 0,C 180,E1 -19060.213,E2 -19060.213} C_VEL
LIN {X 0,Y 249.237,Z 272.432,A -85,B 0,C 180,E1 -19063.624,E2 -19063.624} C_VEL
LIN {X 0,Y 249.239,Z 272.426,A -85,B 0,C 180,E1 -19068.618,E2 -19068.618} C_VEL
LIN {X 0,Y 249.45,Z 272.406,A -85,B 0,C 180,E1 -19071.904,E2 -19071.904} C_VEL
LIN {X 0,Y 249.292,Z 272.43,A -85,B 0,C 180,E1 -19075.15,E2 -19075.15} C_VEL
LIN {X 0,Y 249.672,Z 272.385,A -85,B 0,C 180,E1 -19078.389,E2 -19078.389} C_VEL
LIN {X 0,Y 249.673,Z 272.38,A -85,B 0,C 180,E1 -19081.615,E2 -19081.615} C_VEL
LIN {X 0,Y 249.459,Z 272.405,A -85,B 0,C 180,E1 -19086.472,E2 -19086.472} C_VEL
LIN {X 0,Y 249.387,Z 272.418,A -85,B 0,C 180,E1 -19089.737,E2 -19089.737} C_VEL
LIN {X 0,Y 249.197,Z 272.441,A -85,B 0,C 180,E1 -19094.706,E2 -19094.706} C_VEL
LIN {X 0,Y 249.135,Z 272.445,A -85,B 0,C 180,E1 -19098.08,E2 -19098.08} C_VEL
LIN {X 0,Y 249.087,Z 272.456,A -85,B 0,C 180,E1 -19101.52,E2 -19101.52} C_VEL
LIN {X 0,Y 249.131,Z 272.454,A -85,B 0,C 180,E1 -19105.483,E2 -19105.483} C_VEL
LIN {X 0,Y 249.081,Z 272.455,A -85,B 0,C 180,E1 -19108.993,E2 -19108.993} C_VEL
LIN {X 0,Y 249.032,Z 272.464,A -85,B 0,C 180,E1 -19112.428,E2 -19112.428} C_VEL
LIN {X 0,Y 249.032,Z 272.462,A -85,B 0,C 180,E1 -19116.347,E2 -19116.347} C_VEL
LIN {X 0,Y 249.032,Z 272.464,A -85,B 0,C 180,E1 -19118.174,E2 -19118.174} C_VEL
LIN {X 0,Y 248.326,Z 272.553,A -85,B 0,C 180,E1 -19119.526,E2 -19119.526} C_VEL
LIN {X 0,Y 245.421,Z 272.915,A -85,B 0,C 180,E1 -19121.729,E2 -19121.729} C_VEL
LIN {X 0,Y 242.66,Z 273.606,A -85,B 0,C 180,E1 -19123.968,E2 -19123.968} C_VEL
LIN {X 0,Y 242.198,Z 274.573,A -85,B 0,C 180,E1 -19125.343,E2 -19125.343} C_VEL
LIN {X 0,Y 242.82,Z 277.926,A -85,B 0,C 180,E1 -19128.812,E2 -19128.812} C_VEL
LIN {X 0,Y 243.271,Z 280.397,A -85,B 0,C 180,E1 -19131.265,E2 -19131.265} C_VEL
LIN {X 0,Y 243.397,Z 283.225,A -85,B 0,C 180,E1 -19133.951,E2 -19133.951} C_VEL
LIN {X 0,Y 242.757,Z 286.697,A -85,B 0,C 180,E1 -19137.098,E2 -19137.098} C_VEL
LIN {X 0,Y 241.621,Z 292.951,A -85,B 0,C 180,E1 -19142.605,E2 -19142.605} C_VEL
LIN {X 0,Y 244.12,Z 305.82,A -85,B 0,C 180,E1 -19143.582,E2 -19143.582} C_VEL
LIN {X 0,Y 245.989,Z 318.362,A -85,B 0,C 180,E1 -19144.812,E2 -19144.812} C_VEL
LIN {X 0,Y 247.372,Z 330.972,A -85,B 0,C 180,E1 -19146.343,E2 -19146.343} C_VEL
LIN {X 0,Y 248.043,Z 341.921,A -85,B 0,C 180,E1 -19147.95,E2 -19147.95} C_VEL
LIN {X 0,Y 246.228,Z 352.66,A -85,B 0,C 180,E1 -19149.752,E2 -19149.752} C_VEL
LIN {X 0,Y 244.434,Z 363.276,A -85,B 0,C 180,E1 -19151.996,E2 -19151.996} C_VEL
LIN {X 0,Y 242.87,Z 372.491,A -85,B 0,C 180,E1 -19154.474,E2 -19154.474} C_VEL
LIN {X 0,Y 241.474,Z 379.885,A -85,B 0,C 180,E1 -19156.964,E2 -19156.964} C_VEL
LIN {X 0,Y 240.794,Z 384.918,A -85,B 0,C 180,E1 -19159.064,E2 -19159.064} C_VEL
LIN {X 0,Y 240.21,Z 389.78,A -85,B 0,C 180,E1 -19161.588,E2 -19161.588} C_VEL
LIN {X 0,Y 239.897,Z 393.49,A -85,B 0,C 180,E1 -19164.115,E2 -19164.115} C_VEL
LIN {X 0,Y 239.813,Z 396.154,A -85,B 0,C 180,E1 -19166.64,E2 -19166.64} C_VEL
LIN {X 0,Y 239.868,Z 397.395,A -85,B 0,C 180,E1 -19168.321,E2 -19168.321} C_VEL
LIN {X 0,Y 239.916,Z 398.222,A -85,B 0,C 180,E1 -19170,E2 -19170} C_VEL
LIN {X 0,Y 239.834,Z 398.598,A -85,B 0,C 180,E1 -19171.679,E2 -19171.679} C_VEL
LIN {X 0,Y 239.806,Z 398.179,A -85,B 0,C 180,E1 -19175.044,E2 -19175.044} C_VEL
LIN {X 0,Y 239.961,Z 397.395,A -85,B 0,C 180,E1 -19176.727,E2 -19176.727} C_VEL
LIN {X 0,Y 240.238,Z 396.181,A -85,B 0,C 180,E1 -19178.411,E2 -19178.411} C_VEL
LIN {X 0,Y 241.282,Z 392.53,A -85,B 0,C 180,E1 -19181.764,E2 -19181.764} C_VEL
LIN {X 0,Y 242.512,Z 388.637,A -85,B 0,C 180,E1 -19184.26,E2 -19184.26} C_VEL
LIN {X 0,Y 244.337,Z 383.65,A -85,B 0,C 180,E1 -19186.716,E2 -19186.716} C_VEL
LIN {X 0,Y 246.552,Z 377.469,A -85,B 0,C 180,E1 -19189.135,E2 -19189.135} C_VEL
LIN {X 0,Y 248.414,Z 371.324,A -85,B 0,C 180,E1 -19191.113,E2 -19191.113} C_VEL
LIN {X 0,Y 250.808,Z 363.805,A -85,B 0,C 180,E1 -19193.097,E2 -19193.097} C_VEL
LIN {X 0,Y 254.011,Z 353.902,A -85,B 0,C 180,E1 -19195.175,E2 -19195.175} C_VEL
LIN {X 0,Y 255.185,Z 349.737,A -85,B 0,C 180,E1 -19195.925,E2 -19195.925} C_VEL
LIN {X 0,Y 255.596,Z 339.361,A -85,B 0,C 180,E1 -19197.867,E2 -19197.867} C_VEL
LIN {X 0,Y 255.059,Z 330.097,A -85,B 0,C 180,E1 -19199.493,E2 -19199.493} C_VEL
LIN {X 0,Y 253.187,Z 318.648,A -85,B 0,C 180,E1 -19201.407,E2 -19201.407} C_VEL
LIN {X 0,Y 250.441,Z 307.821,A -85,B 0,C 180,E1 -19203.185,E2 -19203.185} C_VEL
LIN {X 0,Y 247.3,Z 299.207,A -85,B 0,C 180,E1 -19204.671,E2 -19204.671} C_VEL
LIN {X 0,Y 245.693,Z 295.125,A -85,B 0,C 180,E1 -19205.354,E2 -19205.354} C_VEL
LIN {X 0,Y 244.26,Z 291.795,A -85,B 0,C 180,E1 -19205.949,E2 -19205.949} C_VEL
LIN {X 0,Y 244.098,Z 290.798,A -85,B 0,C 180,E1 -19206.107,E2 -19206.107} C_VEL
LIN {X 0,Y 244.241,Z 288.061,A -85,B 0,C 180,E1 -19209.274,E2 -19209.274} C_VEL
LIN {X 0,Y 244.089,Z 286.291,A -85,B 0,C 180,E1 -19211.527,E2 -19211.527} C_VEL
LIN {X 0,Y 243.861,Z 284.548,A -85,B 0,C 180,E1 -19213.903,E2 -19213.903} C_VEL
LIN {X 0,Y 243.445,Z 281.63,A -85,B 0,C 180,E1 -19218.393,E2 -19218.393} C_VEL
LIN {X 0,Y 243.055,Z 279.333,A -85,B 0,C 180,E1 -19222.609,E2 -19222.609} C_VEL
LIN {X 0,Y 242.71,Z 277.568,A -85,B 0,C 180,E1 -19226.619,E2 -19226.619} C_VEL
LIN {X 0,Y 242.561,Z 276.219,A -85,B 0,C 180,E1 -19230.489,E2 -19230.489} C_VEL
LIN {X 0,Y 242.423,Z 275.287,A -85,B 0,C 180,E1 -19234.222,E2 -19234.222} C_VEL
LIN {X 0,Y 242.292,Z 274.693,A -85,B 0,C 180,E1 -19238.153,E2 -19238.153} C_VEL
LIN {X 0,Y 242.374,Z 274.456,A -85,B 0,C 180,E1 -19243.142,E2 -19243.142} C_VEL
LIN {X 0,Y 242.498,Z 274.859,A -85,B 0,C 180,E1 -19248.293,E2 -19248.293} C_VEL
LIN {X 0,Y 242.756,Z 275.428,A -85,B 0,C 180,E1 -19251.675,E2 -19251.675} C_VEL
LIN {X 0,Y 243.026,Z 276.775,A -85,B 0,C 180,E1 -19256.682,E2 -19256.682} C_VEL
LIN {X 0,Y 243.492,Z 277.896,A -85,B 0,C 180,E1 -19259.998,E2 -19259.998} C_VEL
LIN {X 0,Y 243.38,Z 279.356,A -85,B 0,C 180,E1 -19263.309,E2 -19263.309} C_VEL
LIN {X 0,Y 243.416,Z 281.154,A -85,B 0,C 180,E1 -19266.925,E2 -19266.925} C_VEL
LIN {X 0,Y 243.402,Z 282.901,A -85,B 0,C 180,E1 -19269.869,E2 -19269.869} C_VEL
LIN {X 0,Y 244.424,Z 285.826,A -85,B 0,C 180,E1 -19270.346,E2 -19270.346} C_VEL
LIN {X 0,Y 245.769,Z 288.087,A -85,B 0,C 180,E1 -19270.859,E2 -19270.859} C_VEL
LIN {X 0,Y 250.563,Z 298.902,A -85,B 0,C 180,E1 -19272.965,E2 -19272.965} C_VEL
LIN {X 0,Y 254.317,Z 310.361,A -85,B 0,C 180,E1 -19275.107,E2 -19275.107} C_VEL
LIN {X 0,Y 256.62,Z 321.183,A -85,B 0,C 180,E1 -19277.12,E2 -19277.12} C_VEL
LIN {X 0,Y 257.519,Z 329.433,A -85,B 0,C 180,E1 -19278.701,E2 -19278.701} C_VEL
LIN {X 0,Y 257.637,Z 333.583,A -85,B 0,C 180,E1 -19279.52,E2 -19279.52} C_VEL
LIN {X 0,Y 254.64,Z 344.404,A -85,B 0,C 180,E1 -19281.448,E2 -19281.448} C_VEL
LIN {X 0,Y 251.789,Z 353.499,A -85,B 0,C 180,E1 -19283.483,E2 -19283.483} C_VEL
LIN {X 0,Y 249,Z 361.753,A -85,B 0,C 180,E1 -19285.8,E2 -19285.8} C_VEL
LIN {X 0,Y 246.287,Z 369.157,A -85,B 0,C 180,E1 -19288.473,E2 -19288.473} C_VEL
LIN {X 0,Y 244.073,Z 375.002,A -85,B 0,C 180,E1 -19291.216,E2 -19291.216} C_VEL
LIN {X 0,Y 242.745,Z 378.542,A -85,B 0,C 180,E1 -19293.37,E2 -19293.37} C_VEL
LIN {X 0,Y 241.187,Z 382.484,A -85,B 0,C 180,E1 -19296.678,E2 -19296.678} C_VEL
LIN {X 0,Y 240.736,Z 383.561,A -85,B 0,C 180,E1 -19297.981,E2 -19297.981} C_VEL
LIN {X 0,Y 240.057,Z 384.911,A -85,B 0,C 180,E1 -19300.433,E2 -19300.433} C_VEL
LIN {X 0,Y 239.632,Z 385.409,A -85,B 0,C 180,E1 -19302.846,E2 -19302.846} C_VEL
LIN {X 0,Y 239.448,Z 385.118,A -85,B 0,C 180,E1 -19305.219,E2 -19305.219} C_VEL
LIN {X 0,Y 239.409,Z 384.092,A -85,B 0,C 180,E1 -19307.533,E2 -19307.533} C_VEL
LIN {X 0,Y 239.764,Z 381.125,A -85,B 0,C 180,E1 -19310.936,E2 -19310.936} C_VEL
LIN {X 0,Y 240.24,Z 378.098,A -85,B 0,C 180,E1 -19313.241,E2 -19313.241} C_VEL
LIN {X 0,Y 240.866,Z 374.041,A -85,B 0,C 180,E1 -19315.611,E2 -19315.611} C_VEL
LIN {X 0,Y 241.886,Z 367.71,A -85,B 0,C 180,E1 -19318.468,E2 -19318.468} C_VEL
LIN {X 0,Y 243.201,Z 360.361,A -85,B 0,C 180,E1 -19321.051,E2 -19321.051} C_VEL
LIN {X 0,Y 244.8,Z 351.249,A -85,B 0,C 180,E1 -19323.578,E2 -19323.578} C_VEL
LIN {X 0,Y 246.544,Z 341.176,A -85,B 0,C 180,E1 -19325.804,E2 -19325.804} C_VEL
LIN {X 0,Y 248.482,Z 329.813,A -85,B 0,C 180,E1 -19327.773,E2 -19327.773} C_VEL
LIN {X 0,Y 249.404,Z 323.08,A -85,B 0,C 180,E1 -19328.752,E2 -19328.752} C_VEL
LIN {X 0,Y 248.153,Z 313.279,A -85,B 0,C 180,E1 -19330.133,E2 -19330.133} C_VEL
LIN {X 0,Y 246.093,Z 301.665,A -85,B 0,C 180,E1 -19331.518,E2 -19331.518} C_VEL
LIN {X 0,Y 243.078,Z 288.439,A -85,B 0,C 180,E1 -19332.806,E2 -19332.806} C_VEL
LIN {X 0,Y 241.148,Z 280.536,A -85,B 0,C 180,E1 -19333.43,E2 -19333.43} C_VEL
LIN {X 0,Y 241.623,Z 276.363,A -85,B 0,C 180,E1 -19338.253,E2 -19338.253} C_VEL
LIN {X 0,Y 242.235,Z 273.312,A -85,B 0,C 180,E1 -19342.079,E2 -19342.079} C_VEL
LIN {X 0,Y 242.225,Z 273.313,A -85,B 0,C 180,E1 -19345.007,E2 -19345.007} C_VEL
LIN {X 0,Y 242.627,Z 273.262,A -85,B 0,C 180,E1 -19348.34,E2 -19348.34} C_VEL
LIN {X 0,Y 242.63,Z 273.26,A -85,B 0,C 180,E1 -19351.66,E2 -19351.66} C_VEL
LIN {X 0,Y 242.425,Z 273.29,A -85,B 0,C 180,E1 -19356.659,E2 -19356.659} C_VEL
LIN {X 0,Y 242.336,Z 273.299,A -85,B 0,C 180,E1 -19360.021,E2 -19360.021} C_VEL
LIN {X 0,Y 242.158,Z 273.319,A -85,B 0,C 180,E1 -19365.141,E2 -19365.141} C_VEL
LIN {X 0,Y 242.071,Z 273.328,A -85,B 0,C 180,E1 -19368.624,E2 -19368.624} C_VEL
LIN {X 0,Y 242.043,Z 273.336,A -85,B 0,C 180,E1 -19372.177,E2 -19372.177} C_VEL
LIN {X 0,Y 242.058,Z 273.331,A -85,B 0,C 180,E1 -19375.839,E2 -19375.839} C_VEL
LIN {X 0,Y 241.998,Z 273.335,A -85,B 0,C 180,E1 -19379.584,E2 -19379.584} C_VEL
LIN {X 0,Y 241.983,Z 273.343,A -85,B 0,C 180,E1 -19383.492,E2 -19383.492} C_VEL
LIN {X 0,Y 242.005,Z 273.338,A -85,B 0,C 180,E1 -19387.578,E2 -19387.578} C_VEL
LIN {X 0,Y 242.028,Z 273.324,A -85,B 0,C 180,E1 -19391.902,E2 -19391.902} C_VEL
LIN {X 0,Y 242.016,Z 273.334,A -85,B 0,C 180,E1 -19396.55,E2 -19396.55} C_VEL
LIN {X 0,Y 242.003,Z 273.338,A -85,B 0,C 180,E1 -19400.293,E2 -19400.293} C_VEL
LIN {X 0,Y 242.029,Z 273.332,A -85,B 0,C 180,E1 -19404.499,E2 -19404.499} C_VEL
LIN {X 0,Y 241.969,Z 273.33,A -85,B 0,C 180,E1 -19408.482,E2 -19408.482} C_VEL
LIN {X 0,Y 242.002,Z 273.33,A -85,B 0,C 180,E1 -19412.314,E2 -19412.314} C_VEL
LIN {X 0,Y 242.051,Z 273.331,A -85,B 0,C 180,E1 -19416.018,E2 -19416.018} C_VEL
LIN {X 0,Y 242.032,Z 273.334,A -85,B 0,C 180,E1 -19419.61,E2 -19419.61} C_VEL
LIN {X 0,Y 242.158,Z 273.314,A -85,B 0,C 180,E1 -19423.28,E2 -19423.28} C_VEL
LIN {X 0,Y 242.175,Z 273.303,A -85,B 0,C 180,E1 -19428.281,E2 -19428.281} C_VEL
LIN {X 0,Y 242.396,Z 273.283,A -85,B 0,C 180,E1 -19431.667,E2 -19431.667} C_VEL
LIN {X 0,Y 242.253,Z 273.307,A -85,B 0,C 180,E1 -19435.009,E2 -19435.009} C_VEL
LIN {X 0,Y 242.633,Z 273.262,A -85,B 0,C 180,E1 -19438.342,E2 -19438.342} C_VEL
LIN {X 0,Y 242.633,Z 273.257,A -85,B 0,C 180,E1 -19441.662,E2 -19441.662} C_VEL
LIN {X 0,Y 242.431,Z 273.279,A -85,B 0,C 180,E1 -19446.661,E2 -19446.661} C_VEL
LIN {X 0,Y 242.313,Z 273.302,A -85,B 0,C 180,E1 -19450.024,E2 -19450.024} C_VEL
LIN {X 0,Y 242.156,Z 273.318,A -85,B 0,C 180,E1 -19455.143,E2 -19455.143} C_VEL
LIN {X 0,Y 242.07,Z 273.323,A -85,B 0,C 180,E1 -19458.626,E2 -19458.626} C_VEL
LIN {X 0,Y 242.013,Z 273.338,A -85,B 0,C 180,E1 -19462.182,E2 -19462.182} C_VEL
LIN {X 0,Y 242.068,Z 273.33,A -85,B 0,C 180,E1 -19465.84,E2 -19465.84} C_VEL
LIN {X 0,Y 242.03,Z 273.337,A -85,B 0,C 180,E1 -19469.582,E2 -19469.582} C_VEL
LIN {X 0,Y 241.982,Z 273.344,A -85,B 0,C 180,E1 -19473.494,E2 -19473.494} C_VEL
LIN {X 0,Y 241.989,Z 273.343,A -85,B 0,C 180,E1 -19477.584,E2 -19477.584} C_VEL
LIN {X 0,Y 241.941,Z 273.348,A -85,B 0,C 180,E1 -19481.924,E2 -19481.924} C_VEL
LIN {X 0,Y 242.021,Z 273.479,A -85,B 0,C 180,E1 -19484.184,E2 -19484.184} C_VEL
LIN {X 0,Y 242.198,Z 274.573,A -85,B 0,C 180,E1 -19485.343,E2 -19485.343} C_VEL
LIN {X 0,Y 241.829,Z 275.954,A -85,B 0,C 180,E1 -19486.696,E2 -19486.696} C_VEL
LIN {X 0,Y 239.477,Z 278.48,A -85,B 0,C 180,E1 -19488.903,E2 -19488.903} C_VEL
LIN {X 0,Y 236.623,Z 281.589,A -85,B 0,C 180,E1 -19491.613,E2 -19491.613} C_VEL
LIN {X 0,Y 236.327,Z 282.58,A -85,B 0,C 180,E1 -19492.548,E2 -19492.548} C_VEL
LIN {X 0,Y 236.055,Z 285.73,A -85,B 0,C 180,E1 -19495.551,E2 -19495.551} C_VEL
LIN {X 0,Y 234.918,Z 290.799,A -85,B 0,C 180,E1 -19500.183,E2 -19500.183} C_VEL
LIN {X 0,Y 234.627,Z 292.774,A -85,B 0,C 180,E1 -19501.969,E2 -19501.969} C_VEL
LIN {X 0,Y 237.142,Z 305.705,A -85,B 0,C 180,E1 -19502.995,E2 -19502.995} C_VEL
LIN {X 0,Y 239.117,Z 318.681,A -85,B 0,C 180,E1 -19504.315,E2 -19504.315} C_VEL
LIN {X 0,Y 240.407,Z 330.882,A -85,B 0,C 180,E1 -19505.841,E2 -19505.841} C_VEL
LIN {X 0,Y 241.147,Z 341.864,A -85,B 0,C 180,E1 -19507.511,E2 -19507.511} C_VEL
LIN {X 0,Y 239.343,Z 352.584,A -85,B 0,C 180,E1 -19509.368,E2 -19509.368} C_VEL
LIN {X 0,Y 237.496,Z 362.889,A -85,B 0,C 180,E1 -19511.603,E2 -19511.603} C_VEL
LIN {X 0,Y 235.969,Z 371.686,A -85,B 0,C 180,E1 -19514.008,E2 -19514.008} C_VEL
LIN {X 0,Y 234.53,Z 379.182,A -85,B 0,C 180,E1 -19516.571,E2 -19516.571} C_VEL
LIN {X 0,Y 233.528,Z 386.113,A -85,B 0,C 180,E1 -19519.597,E2 -19519.597} C_VEL
LIN {X 0,Y 233.009,Z 390.659,A -85,B 0,C 180,E1 -19522.199,E2 -19522.199} C_VEL
LIN {X 0,Y 232.71,Z 394.609,A -85,B 0,C 180,E1 -19525.309,E2 -19525.309} C_VEL
LIN {X 0,Y 232.779,Z 397.058,A -85,B 0,C 180,E1 -19528.27,E2 -19528.27} C_VEL
LIN {X 0,Y 232.848,Z 397.93,A -85,B 0,C 180,E1 -19530,E2 -19530} C_VEL
LIN {X 0,Y 232.745,Z 398.374,A -85,B 0,C 180,E1 -19531.73,E2 -19531.73} C_VEL
LIN {X 0,Y 232.736,Z 398.033,A -85,B 0,C 180,E1 -19535.197,E2 -19535.197} C_VEL
LIN {X 0,Y 233.206,Z 396.149,A -85,B 0,C 180,E1 -19538.666,E2 -19538.666} C_VEL
LIN {X 0,Y 234.322,Z 392.584,A -85,B 0,C 180,E1 -19542.119,E2 -19542.119} C_VEL
LIN {X 0,Y 235.632,Z 388.797,A -85,B 0,C 180,E1 -19544.685,E2 -19544.685} C_VEL
LIN {X 0,Y 237.549,Z 383.933,A -85,B 0,C 180,E1 -19547.208,E2 -19547.208} C_VEL
LIN {X 0,Y 239.852,Z 377.863,A -85,B 0,C 180,E1 -19549.691,E2 -19549.691} C_VEL
LIN {X 0,Y 242.321,Z 370.408,A -85,B 0,C 180,E1 -19552.15,E2 -19552.15} C_VEL
LIN {X 0,Y 244.976,Z 362.852,A -85,B 0,C 180,E1 -19554.129,E2 -19554.129} C_VEL
LIN {X 0,Y 248.314,Z 352.78,A -85,B 0,C 180,E1 -19556.246,E2 -19556.246} C_VEL
LIN {X 0,Y 248.928,Z 349.733,A -85,B 0,C 180,E1 -19556.854,E2 -19556.854} C_VEL
LIN {X 0,Y 249.384,Z 339.521,A -85,B 0,C 180,E1 -19558.86,E2 -19558.86} C_VEL
LIN {X 0,Y 248.697,Z 329.068,A -85,B 0,C 180,E1 -19560.774,E2 -19560.774} C_VEL
LIN {X 0,Y 246.835,Z 317.987,A -85,B 0,C 180,E1 -19562.749,E2 -19562.749} C_VEL
LIN {X 0,Y 244.192,Z 308.201,A -85,B 0,C 180,E1 -19564.501,E2 -19564.501} C_VEL
LIN {X 0,Y 240.818,Z 298.979,A -85,B 0,C 180,E1 -19566.241,E2 -19566.241} C_VEL
LIN {X 0,Y 239.24,Z 295.257,A -85,B 0,C 180,E1 -19566.963,E2 -19566.963} C_VEL
LIN {X 0,Y 237.585,Z 292.092,A -85,B 0,C 180,E1 -19567.66,E2 -19567.66} C_VEL
LIN {X 0,Y 237.203,Z 290.51,A -85,B 0,C 180,E1 -19567.917,E2 -19567.917} C_VEL
LIN {X 0,Y 237.14,Z 288.315,A -85,B 0,C 180,E1 -19570.692,E2 -19570.692} C_VEL
LIN {X 0,Y 236.819,Z 285.552,A -85,B 0,C 180,E1 -19574.58,E2 -19574.58} C_VEL
LIN {X 0,Y 236.436,Z 282.732,A -85,B 0,C 180,E1 -19579.158,E2 -19579.158} C_VEL
LIN {X 0,Y 236.074,Z 280.524,A -85,B 0,C 180,E1 -19583.492,E2 -19583.492} C_VEL
LIN {X 0,Y 235.76,Z 278.877,A -85,B 0,C 180,E1 -19587.547,E2 -19587.547} C_VEL
LIN {X 0,Y 235.597,Z 277.635,A -85,B 0,C 180,E1 -19591.489,E2 -19591.489} C_VEL
LIN {X 0,Y 235.454,Z 276.806,A -85,B 0,C 180,E1 -19595.297,E2 -19595.297} C_VEL
LIN {X 0,Y 235.367,Z 276.336,A -85,B 0,C 180,E1 -19599.001,E2 -19599.001} C_VEL
LIN {X 0,Y 235.455,Z 276.164,A -85,B 0,C 180,E1 -19602.771,E2 -19602.771} C_VEL
LIN {X 0,Y 235.562,Z 276.488,A -85,B 0,C 180,E1 -19607.943,E2 -19607.943} C_VEL
LIN {X 0,Y 235.837,Z 277.012,A -85,B 0,C 180,E1 -19611.429,E2 -19611.429} C_VEL
LIN {X 0,Y 236.085,Z 278.318,A -85,B 0,C 180,E1 -19616.585,E2 -19616.585} C_VEL
LIN {X 0,Y 236.568,Z 279.411,A -85,B 0,C 180,E1 -19619.998,E2 -19619.998} C_VEL
LIN {X 0,Y 236.441,Z 280.868,A -85,B 0,C 180,E1 -19623.406,E2 -19623.406} C_VEL
LIN {X 0,Y 236.437,Z 283.12,A -85,B 0,C 180,E1 -19628.007,E2 -19628.007} C_VEL
LIN {X 0,Y 237.662,Z 286.275,A -85,B 0,C 180,E1 -19628.608,E2 -19628.608} C_VEL
LIN {X 0,Y 239.277,Z 288.603,A -85,B 0,C 180,E1 -19629.241,E2 -19629.241} C_VEL
LIN {X 0,Y 243.144,Z 297.068,A -85,B 0,C 180,E1 -19631.075,E2 -19631.075} C_VEL
LIN {X 0,Y 246.908,Z 307.207,A -85,B 0,C 180,E1 -19633.16,E2 -19633.16} C_VEL
LIN {X 0,Y 249.442,Z 316.954,A -85,B 0,C 180,E1 -19635.105,E2 -19635.105} C_VEL
LIN {X 0,Y 251.033,Z 326.853,A -85,B 0,C 180,E1 -19637.093,E2 -19637.093} C_VEL
LIN {X 0,Y 251.494,Z 334.415,A -85,B 0,C 180,E1 -19638.659,E2 -19638.659} C_VEL
LIN {X 0,Y 249.074,Z 343.279,A -85,B 0,C 180,E1 -19640.282,E2 -19640.282} C_VEL
LIN {X 0,Y 245.852,Z 353.085,A -85,B 0,C 180,E1 -19642.486,E2 -19642.486} C_VEL
LIN {X 0,Y 242.968,Z 361.128,A -85,B 0,C 180,E1 -19644.743,E2 -19644.743} C_VEL
LIN {X 0,Y 240.063,Z 368.702,A -85,B 0,C 180,E1 -19647.455,E2 -19647.455} C_VEL
LIN {X 0,Y 237.696,Z 374.521,A -85,B 0,C 180,E1 -19650.172,E2 -19650.172} C_VEL
LIN {X 0,Y 235.631,Z 379.604,A -85,B 0,C 180,E1 -19653.372,E2 -19653.372} C_VEL
LIN {X 0,Y 234.37,Z 382.469,A -85,B 0,C 180,E1 -19655.941,E2 -19655.941} C_VEL
LIN {X 0,Y 233.246,Z 384.776,A -85,B 0,C 180,E1 -19659.251,E2 -19659.251} C_VEL
LIN {X 0,Y 232.716,Z 385.551,A -85,B 0,C 180,E1 -19661.633,E2 -19661.633} C_VEL
LIN {X 0,Y 232.399,Z 385.533,A -85,B 0,C 180,E1 -19664.067,E2 -19664.067} C_VEL
LIN {X 0,Y 232.316,Z 384.721,A -85,B 0,C 180,E1 -19666.552,E2 -19666.552} C_VEL
LIN {X 0,Y 232.398,Z 383.026,A -85,B 0,C 180,E1 -19669.112,E2 -19669.112} C_VEL
LIN {X 0,Y 232.812,Z 380.371,A -85,B 0,C 180,E1 -19671.705,E2 -19671.705} C_VEL
LIN {X 0,Y 233.423,Z 376.558,A -85,B 0,C 180,E1 -19674.379,E2 -19674.379} C_VEL
LIN {X 0,Y 234.327,Z 370.945,A -85,B 0,C 180,E1 -19677.327,E2 -19677.327} C_VEL
LIN {X 0,Y 235.465,Z 364.538,A -85,B 0,C 180,E1 -19679.943,E2 -19679.943} C_VEL
LIN {X 0,Y 236.769,Z 357.527,A -85,B 0,C 180,E1 -19682.242,E2 -19682.242} C_VEL
LIN {X 0,Y 238.51,Z 348.145,A -85,B 0,C 180,E1 -19684.708,E2 -19684.708} C_VEL
LIN {X 0,Y 240.176,Z 338.592,A -85,B 0,C 180,E1 -19686.733,E2 -19686.733} C_VEL
LIN {X 0,Y 241.952,Z 327.999,A -85,B 0,C 180,E1 -19688.538,E2 -19688.538} C_VEL
LIN {X 0,Y 242.508,Z 323.098,A -85,B 0,C 180,E1 -19689.258,E2 -19689.258} C_VEL
LIN {X 0,Y 240.75,Z 310.701,A -85,B 0,C 180,E1 -19691.013,E2 -19691.013} C_VEL
LIN {X 0,Y 238.307,Z 298.06,A -85,B 0,C 180,E1 -19692.5,E2 -19692.5} C_VEL
LIN {X 0,Y 235.105,Z 284.849,A -85,B 0,C 180,E1 -19693.745,E2 -19693.745} C_VEL
LIN {X 0,Y 234.193,Z 280.712,A -85,B 0,C 180,E1 -19694.093,E2 -19694.093} C_VEL
LIN {X 0,Y 234.748,Z 276.054,A -85,B 0,C 180,E1 -19699.652,E2 -19699.652} C_VEL
LIN {X 0,Y 235.207,Z 274.187,A -85,B 0,C 180,E1 -19702.057,E2 -19702.057} C_VEL
LIN {X 0,Y 235.586,Z 274.139,A -85,B 0,C 180,E1 -19708.291,E2 -19708.291} C_VEL
LIN {X 0,Y 235.59,Z 274.138,A -85,B 0,C 180,E1 -19711.71,E2 -19711.71} C_VEL
LIN {X 0,Y 235.396,Z 274.164,A -85,B 0,C 180,E1 -19716.859,E2 -19716.859} C_VEL
LIN {X 0,Y 235.244,Z 274.181,A -85,B 0,C 180,E1 -19720.326,E2 -19720.326} C_VEL
LIN {X 0,Y 235.105,Z 274.198,A -85,B 0,C 180,E1 -19725.607,E2 -19725.607} C_VEL
LIN {X 0,Y 235.011,Z 274.206,A -85,B 0,C 180,E1 -19729.205,E2 -19729.205} C_VEL
LIN {X 0,Y 234.974,Z 274.214,A -85,B 0,C 180,E1 -19732.881,E2 -19732.881} C_VEL
LIN {X 0,Y 234.959,Z 274.21,A -85,B 0,C 180,E1 -19736.658,E2 -19736.658} C_VEL
LIN {X 0,Y 234.914,Z 274.218,A -85,B 0,C 180,E1 -19740.57,E2 -19740.57} C_VEL
LIN {X 0,Y 234.952,Z 274.217,A -85,B 0,C 180,E1 -19744.634,E2 -19744.634} C_VEL
LIN {X 0,Y 234.958,Z 274.212,A -85,B 0,C 180,E1 -19748.953,E2 -19748.953} C_VEL
LIN {X 0,Y 234.988,Z 274.204,A -85,B 0,C 180,E1 -19753.462,E2 -19753.462} C_VEL
LIN {X 0,Y 234.988,Z 274.209,A -85,B 0,C 180,E1 -19756.541,E2 -19756.541} C_VEL
LIN {X 0,Y 234.948,Z 274.22,A -85,B 0,C 180,E1 -19761.088,E2 -19761.088} C_VEL
LIN {X 0,Y 234.953,Z 274.211,A -85,B 0,C 180,E1 -19765.369,E2 -19765.369} C_VEL
LIN {X 0,Y 234.963,Z 274.2,A -85,B 0,C 180,E1 -19770.159,E2 -19770.159} C_VEL
LIN {X 0,Y 234.988,Z 274.207,A -85,B 0,C 180,E1 -19773.796,E2 -19773.796} C_VEL
LIN {X 0,Y 235.006,Z 274.212,A -85,B 0,C 180,E1 -19778.972,E2 -19778.972} C_VEL
LIN {X 0,Y 235.091,Z 274.195,A -85,B 0,C 180,E1 -19783.061,E2 -19783.061} C_VEL
